LIN {X 0,Y 720.158,Z 171.461,A -85,B 0,C 180,E1 33611.893,E2 33611.893} C_VEL
LIN {X 0,Y 720.133,Z 171.461,A -85,B 0,C 180,E1 33608.963,E2 33608.963} C_VEL
LIN {X 0,Y 720.115,Z 171.46,A -85,B 0,C 180,E1 33606.555,E2 33606.555} C_VEL
LIN {X 0,Y 720.175,Z 171.461,A -85,B 0,C 180,E1 33603.874,E2 33603.874} C_VEL
LIN {X 0,Y 720.128,Z 171.46,A -85,B 0,C 180,E1 33601.001,E2 33601.001} C_VEL
LIN {X 0,Y 720.115,Z 171.461,A -85,B 0,C 180,E1 33598.618,E2 33598.618} C_VEL
LIN {X 0,Y 720.167,Z 171.46,A -85,B 0,C 180,E1 33596.02,E2 33596.02} C_VEL
LIN {X 0,Y 720.131,Z 171.461,A -85,B 0,C 180,E1 33593.134,E2 33593.134} C_VEL
LIN {X 0,Y 720.115,Z 171.461,A -85,B 0,C 180,E1 33590.734,E2 33590.734} C_VEL
LIN {X 0,Y 720.152,Z 171.461,A -85,B 0,C 180,E1 33588.201,E2 33588.201} C_VEL
LIN {X 0,Y 720.129,Z 171.461,A -85,B 0,C 180,E1 33585.203,E2 33585.203} C_VEL
LIN {X 0,Y 720.114,Z 171.461,A -85,B 0,C 180,E1 33582.834,E2 33582.834} C_VEL
LIN {X 0,Y 720.15,Z 171.461,A -85,B 0,C 180,E1 33580.316,E2 33580.316} C_VEL
LIN {X 0,Y 720.133,Z 171.462,A -85,B 0,C 180,E1 33577.338,E2 33577.338} C_VEL
LIN {X 0,Y 720.114,Z 171.461,A -85,B 0,C 180,E1 33574.938,E2 33574.938} C_VEL
LIN {X 0,Y 720.151,Z 171.462,A -85,B 0,C 180,E1 33572.387,E2 33572.387} C_VEL
LIN {X 0,Y 720.134,Z 171.462,A -85,B 0,C 180,E1 33569.443,E2 33569.443} C_VEL
LIN {X 0,Y 720.113,Z 171.462,A -85,B 0,C 180,E1 33567.056,E2 33567.056} C_VEL
LIN {X 0,Y 720.139,Z 171.461,A -85,B 0,C 180,E1 33564.583,E2 33564.583} C_VEL
LIN {X 0,Y 720.135,Z 171.461,A -85,B 0,C 180,E1 33561.538,E2 33561.538} C_VEL
LIN {X 0,Y 720.116,Z 171.461,A -85,B 0,C 180,E1 33559.036,E2 33559.036} C_VEL
LIN {X 0,Y 720.183,Z 171.461,A -85,B 0,C 180,E1 33556.35,E2 33556.35} C_VEL
LIN {X 0,Y 720.123,Z 171.461,A -85,B 0,C 180,E1 33553.465,E2 33553.465} C_VEL
LIN {X 0,Y 720.118,Z 171.461,A -85,B 0,C 180,E1 33551.043,E2 33551.043} C_VEL
LIN {X 0,Y 720.213,Z 171.46,A -85,B 0,C 180,E1 33548.245,E2 33548.245} C_VEL
LIN {X 0,Y 720.117,Z 171.461,A -85,B 0,C 180,E1 33545.433,E2 33545.433} C_VEL
LIN {X 0,Y 720.125,Z 171.46,A -85,B 0,C 180,E1 33543.001,E2 33543.001} C_VEL
LIN {X 0,Y 720.179,Z 171.46,A -85,B 0,C 180,E1 33540.108,E2 33540.108} C_VEL
LIN {X 0,Y 720.116,Z 171.461,A -85,B 0,C 180,E1 33537.44,E2 33537.44} C_VEL
LIN {X 0,Y 720.139,Z 171.461,A -85,B 0,C 180,E1 33534.918,E2 33534.918} C_VEL
LIN {X 0,Y 720.134,Z 171.461,A -85,B 0,C 180,E1 33531.845,E2 33531.845} C_VEL
LIN {X 0,Y 720.115,Z 171.46,A -85,B 0,C 180,E1 33529.422,E2 33529.422} C_VEL
LIN {X 0,Y 720.149,Z 171.461,A -85,B 0,C 180,E1 33526.914,E2 33526.914} C_VEL
LIN {X 0,Y 720.131,Z 171.46,A -85,B 0,C 180,E1 33523.902,E2 33523.902} C_VEL
LIN {X 0,Y 720.116,Z 171.46,A -85,B 0,C 180,E1 33521.436,E2 33521.436} C_VEL
LIN {X 0,Y 720.193,Z 171.46,A -85,B 0,C 180,E1 33518.725,E2 33518.725} C_VEL
LIN {X 0,Y 720.121,Z 171.453,A -85,B 0,C 180,E1 33515.87,E2 33515.87} C_VEL
LIN {X 0,Y 720.118,Z 171.457,A -85,B 0,C 180,E1 33513.449,E2 33513.449} C_VEL
LIN {X 0,Y 720.211,Z 171.457,A -85,B 0,C 180,E1 33510.611,E2 33510.611} C_VEL
LIN {X 0,Y 720.117,Z 171.447,A -85,B 0,C 180,E1 33507.827,E2 33507.827} C_VEL
LIN {X 0,Y 720.126,Z 171.457,A -85,B 0,C 180,E1 33505.407,E2 33505.407} C_VEL
LIN {X 0,Y 720.166,Z 171.457,A -85,B 0,C 180,E1 33502.446,E2 33502.446} C_VEL
LIN {X 0,Y 720.116,Z 171.46,A -85,B 0,C 180,E1 33499.888,E2 33499.888} C_VEL
LIN {X 0,Y 720.126,Z 171.458,A -85,B 0,C 180,E1 33497.491,E2 33497.491} C_VEL
LIN {X 0,Y 720.167,Z 171.459,A -85,B 0,C 180,E1 33494.555,E2 33494.555} C_VEL
LIN {X 0,Y 720.115,Z 171.457,A -85,B 0,C 180,E1 33491.94,E2 33491.94} C_VEL
LIN {X 0,Y 720.14,Z 171.46,A -85,B 0,C 180,E1 33489.43,E2 33489.43} C_VEL
LIN {X 0,Y 720.136,Z 171.459,A -85,B 0,C 180,E1 33486.377,E2 33486.377} C_VEL
LIN {X 0,Y 720.115,Z 171.46,A -85,B 0,C 180,E1 33483.901,E2 33483.901} C_VEL
LIN {X 0,Y 720.169,Z 171.457,A -85,B 0,C 180,E1 33481.273,E2 33481.273} C_VEL
LIN {X 0,Y 720.126,Z 171.458,A -85,B 0,C 180,E1 33478.334,E2 33478.334} C_VEL
LIN {X 0,Y 720.117,Z 171.458,A -85,B 0,C 180,E1 33475.939,E2 33475.939} C_VEL
LIN {X 0,Y 720.21,Z 171.459,A -85,B 0,C 180,E1 33473.143,E2 33473.143} C_VEL
LIN {X 0,Y 720.12,Z 171.459,A -85,B 0,C 180,E1 33470.3,E2 33470.3} C_VEL
LIN {X 0,Y 720.123,Z 171.458,A -85,B 0,C 180,E1 33467.897,E2 33467.897} C_VEL
LIN {X 0,Y 720.195,Z 171.46,A -85,B 0,C 180,E1 33465.035,E2 33465.035} C_VEL
LIN {X 0,Y 720.117,Z 171.457,A -85,B 0,C 180,E1 33462.297,E2 33462.297} C_VEL
LIN {X 0,Y 720.131,Z 171.46,A -85,B 0,C 180,E1 33459.858,E2 33459.858} C_VEL
LIN {X 0,Y 720.155,Z 171.46,A -85,B 0,C 180,E1 33456.863,E2 33456.863} C_VEL
LIN {X 0,Y 720.117,Z 171.458,A -85,B 0,C 180,E1 33454.292,E2 33454.292} C_VEL
LIN {X 0,Y 720.152,Z 171.451,A -85,B 0,C 180,E1 33451.741,E2 33451.741} C_VEL
LIN {X 0,Y 720.136,Z 171.46,A -85,B 0,C 180,E1 33448.78,E2 33448.78} C_VEL
LIN {X 0,Y 720.116,Z 171.458,A -85,B 0,C 180,E1 33446.357,E2 33446.357} C_VEL
LIN {X 0,Y 720.165,Z 171.456,A -85,B 0,C 180,E1 33443.739,E2 33443.739} C_VEL
LIN {X 0,Y 720.128,Z 171.456,A -85,B 0,C 180,E1 33440.775,E2 33440.775} C_VEL
LIN {X 0,Y 720.117,Z 171.46,A -85,B 0,C 180,E1 33438.416,E2 33438.416} C_VEL
LIN {X 0,Y 720.178,Z 171.459,A -85,B 0,C 180,E1 33435.751,E2 33435.751} C_VEL
LIN {X 0,Y 720.127,Z 171.458,A -85,B 0,C 180,E1 33432.851,E2 33432.851} C_VEL
LIN {X 0,Y 720.119,Z 171.461,A -85,B 0,C 180,E1 33430.456,E2 33430.456} C_VEL
LIN {X 0,Y 720.191,Z 171.446,A -85,B 0,C 180,E1 33427.748,E2 33427.748} C_VEL
LIN {X 0,Y 720.122,Z 171.461,A -85,B 0,C 180,E1 33424.854,E2 33424.854} C_VEL
LIN {X 0,Y 720.122,Z 171.447,A -85,B 0,C 180,E1 33422.404,E2 33422.404} C_VEL
LIN {X 0,Y 720.19,Z 171.751,A -85,B 0,C 180,E1 33421.207,E2 33421.207} C_VEL
LIN {X 0,Y 722.827,Z 180.968,A -85,B 0,C 180,E1 33420.32,E2 33420.32} C_VEL
LIN {X 0,Y 722.315,Z 216.19,A -85,B 0,C 180,E1 33417.535,E2 33417.535} C_VEL
LIN {X 0,Y 722.261,Z 226.415,A -85,B 0,C 180,E1 33416.755,E2 33416.755} C_VEL
LIN {X 0,Y 723.859,Z 234.554,A -85,B 0,C 180,E1 33416.596,E2 33416.596} C_VEL
LIN {X 0,Y 723.073,Z 507.416,A -85,B 0,C 180,E1 33413.694,E2 33413.694} C_VEL
LIN {X 0,Y 722.911,Z 536.198,A -85,B 0,C 180,E1 33413.337,E2 33413.337} C_VEL
LIN {X 0,Y 722.72,Z 557.475,A -85,B 0,C 180,E1 33412.924,E2 33412.924} C_VEL
LIN {X 0,Y 722.482,Z 576.531,A -85,B 0,C 180,E1 33412.43,E2 33412.43} C_VEL
LIN {X 0,Y 722.235,Z 596.799,A -85,B 0,C 180,E1 33411.776,E2 33411.776} C_VEL
LIN {X 0,Y 721.924,Z 617.74,A -85,B 0,C 180,E1 33410.934,E2 33410.934} C_VEL
LIN {X 0,Y 721.584,Z 636.362,A -85,B 0,C 180,E1 33410.032,E2 33410.032} C_VEL
LIN {X 0,Y 721.311,Z 654.533,A -85,B 0,C 180,E1 33409.009,E2 33409.009} C_VEL
LIN {X 0,Y 720.986,Z 673.25,A -85,B 0,C 180,E1 33407.762,E2 33407.762} C_VEL
LIN {X 0,Y 720.714,Z 689.21,A -85,B 0,C 180,E1 33406.521,E2 33406.521} C_VEL
LIN {X 0,Y 720.486,Z 704.756,A -85,B 0,C 180,E1 33405.122,E2 33405.122} C_VEL
LIN {X 0,Y 720.286,Z 719.459,A -85,B 0,C 180,E1 33403.566,E2 33403.566} C_VEL
LIN {X 0,Y 720.163,Z 731.326,A -85,B 0,C 180,E1 33402.1,E2 33402.1} C_VEL
LIN {X 0,Y 720.053,Z 742.382,A -85,B 0,C 180,E1 33400.48,E2 33400.48} C_VEL
LIN {X 0,Y 719.976,Z 751.89,A -85,B 0,C 180,E1 33398.786,E2 33398.786} C_VEL
LIN {X 0,Y 719.946,Z 759.234,A -85,B 0,C 180,E1 33397.179,E2 33397.179} C_VEL
LIN {X 0,Y 719.924,Z 765.17,A -85,B 0,C 180,E1 33395.498,E2 33395.498} C_VEL
LIN {X 0,Y 719.917,Z 769.789,A -85,B 0,C 180,E1 33393.663,E2 33393.663} C_VEL
LIN {X 0,Y 719.919,Z 772.482,A -85,B 0,C 180,E1 33391.91,E2 33391.91} C_VEL
LIN {X 0,Y 719.907,Z 773.462,A -85,B 0,C 180,E1 33390.159,E2 33390.159} C_VEL
LIN {X 0,Y 719.91,Z 772.697,A -85,B 0,C 180,E1 33388.329,E2 33388.329} C_VEL
LIN {X 0,Y 719.908,Z 770.262,A -85,B 0,C 180,E1 33386.577,E2 33386.577} C_VEL
LIN {X 0,Y 719.909,Z 766.362,A -85,B 0,C 180,E1 33384.901,E2 33384.901} C_VEL
LIN {X 0,Y 719.925,Z 760.484,A -85,B 0,C 180,E1 33383.141,E2 33383.141} C_VEL
LIN {X 0,Y 719.965,Z 752.702,A -85,B 0,C 180,E1 33381.375,E2 33381.375} C_VEL
LIN {X 0,Y 720.041,Z 743.892,A -85,B 0,C 180,E1 33379.763,E2 33379.763} C_VEL
LIN {X 0,Y 720.147,Z 732.537,A -85,B 0,C 180,E1 33378.062,E2 33378.062} C_VEL
LIN {X 0,Y 720.262,Z 720.869,A -85,B 0,C 180,E1 33376.597,E2 33376.597} C_VEL
LIN {X 0,Y 720.458,Z 707.3,A -85,B 0,C 180,E1 33375.125,E2 33375.125} C_VEL
LIN {X 0,Y 720.7,Z 691.197,A -85,B 0,C 180,E1 33373.644,E2 33373.644} C_VEL
LIN {X 0,Y 720.947,Z 675.482,A -85,B 0,C 180,E1 33372.404,E2 33372.404} C_VEL
LIN {X 0,Y 721.234,Z 657.839,A -85,B 0,C 180,E1 33371.199,E2 33371.199} C_VEL
LIN {X 0,Y 721.563,Z 638.343,A -85,B 0,C 180,E1 33370.072,E2 33370.072} C_VEL
LIN {X 0,Y 721.867,Z 620.585,A -85,B 0,C 180,E1 33369.196,E2 33369.196} C_VEL
LIN {X 0,Y 722.145,Z 601.277,A -85,B 0,C 180,E1 33368.392,E2 33368.392} C_VEL
LIN {X 0,Y 722.463,Z 579.414,A -85,B 0,C 180,E1 33367.654,E2 33367.654} C_VEL
LIN {X 0,Y 722.691,Z 559.421,A -85,B 0,C 180,E1 33367.121,E2 33367.121} C_VEL
LIN {X 0,Y 722.903,Z 537.995,A -85,B 0,C 180,E1 33366.692,E2 33366.692} C_VEL
LIN {X 0,Y 723.061,Z 510.848,A -85,B 0,C 180,E1 33366.342,E2 33366.342} C_VEL
LIN {X 0,Y 723.844,Z 239.48,A -85,B 0,C 180,E1 33363.457,E2 33363.457} C_VEL
LIN {X 0,Y 723.623,Z 232.466,A -85,B 0,C 180,E1 33363.372,E2 33363.372} C_VEL
LIN {X 0,Y 722.233,Z 225.971,A -85,B 0,C 180,E1 33363.219,E2 33363.219} C_VEL
LIN {X 0,Y 722.711,Z 188.921,A -85,B 0,C 180,E1 33360.315,E2 33360.315} C_VEL
LIN {X 0,Y 722.78,Z 180.457,A -85,B 0,C 180,E1 33359.636,E2 33359.636} C_VEL
LIN {X 0,Y 720.169,Z 171.589,A -85,B 0,C 180,E1 33358.76,E2 33358.76} C_VEL
LIN {X 0,Y 720.136,Z 171.461,A -85,B 0,C 180,E1 33355.788,E2 33355.788} C_VEL
LIN {X 0,Y 720.116,Z 171.457,A -85,B 0,C 180,E1 33353.346,E2 33353.346} C_VEL
LIN {X 0,Y 720.16,Z 171.454,A -85,B 0,C 180,E1 33350.782,E2 33350.782} C_VEL
LIN {X 0,Y 720.132,Z 171.458,A -85,B 0,C 180,E1 33347.855,E2 33347.855} C_VEL
LIN {X 0,Y 720.117,Z 171.46,A -85,B 0,C 180,E1 33345.423,E2 33345.423} C_VEL
LIN {X 0,Y 720.18,Z 171.458,A -85,B 0,C 180,E1 33342.747,E2 33342.747} C_VEL
LIN {X 0,Y 720.127,Z 171.456,A -85,B 0,C 180,E1 33339.849,E2 33339.849} C_VEL
LIN {X 0,Y 720.119,Z 171.46,A -85,B 0,C 180,E1 33337.428,E2 33337.428} C_VEL
LIN {X 0,Y 720.203,Z 171.454,A -85,B 0,C 180,E1 33334.696,E2 33334.696} C_VEL
LIN {X 0,Y 720.12,Z 171.46,A -85,B 0,C 180,E1 33331.827,E2 33331.827} C_VEL
LIN {X 0,Y 720.118,Z 171.455,A -85,B 0,C 180,E1 33329.486,E2 33329.486} C_VEL
LIN {X 0,Y 720.208,Z 171.452,A -85,B 0,C 180,E1 33326.732,E2 33326.732} C_VEL
LIN {X 0,Y 720.121,Z 171.46,A -85,B 0,C 180,E1 33323.919,E2 33323.919} C_VEL
LIN {X 0,Y 720.12,Z 171.457,A -85,B 0,C 180,E1 33321.539,E2 33321.539} C_VEL
LIN {X 0,Y 720.205,Z 171.457,A -85,B 0,C 180,E1 33318.706,E2 33318.706} C_VEL
LIN {X 0,Y 720.118,Z 171.459,A -85,B 0,C 180,E1 33315.958,E2 33315.958} C_VEL
LIN {X 0,Y 720.12,Z 171.458,A -85,B 0,C 180,E1 33313.634,E2 33313.634} C_VEL
LIN {X 0,Y 720.203,Z 171.46,A -85,B 0,C 180,E1 33310.803,E2 33310.803} C_VEL
LIN {X 0,Y 720.118,Z 171.456,A -85,B 0,C 180,E1 33308.062,E2 33308.062} C_VEL
LIN {X 0,Y 720.12,Z 171.46,A -85,B 0,C 180,E1 33305.738,E2 33305.738} C_VEL
LIN {X 0,Y 720.209,Z 171.457,A -85,B 0,C 180,E1 33302.945,E2 33302.945} C_VEL
LIN {X 0,Y 720.119,Z 171.46,A -85,B 0,C 180,E1 33300.159,E2 33300.159} C_VEL
LIN {X 0,Y 720.121,Z 171.457,A -85,B 0,C 180,E1 33297.772,E2 33297.772} C_VEL
LIN {X 0,Y 720.191,Z 171.459,A -85,B 0,C 180,E1 33294.902,E2 33294.902} C_VEL
LIN {X 0,Y 720.119,Z 171.458,A -85,B 0,C 180,E1 33292.26,E2 33292.26} C_VEL
LIN {X 0,Y 720.123,Z 171.46,A -85,B 0,C 180,E1 33289.837,E2 33289.837} C_VEL
LIN {X 0,Y 720.194,Z 171.46,A -85,B 0,C 180,E1 33287.002,E2 33287.002} C_VEL
LIN {X 0,Y 720.116,Z 171.459,A -85,B 0,C 180,E1 33284.29,E2 33284.29} C_VEL
LIN {X 0,Y 720.164,Z 171.459,A -85,B 0,C 180,E1 33283.499,E2 33283.499} C_VEL
LIN {X 0,Y 719.244,Z 171.582,A -85,B 0,C 180,E1 33282.887,E2 33282.887} C_VEL
LIN {X 0,Y 712.687,Z 172.397,A -85,B 0,C 180,E1 33281.126,E2 33281.126} C_VEL
LIN {X 0,Y 712.206,Z 172.449,A -85,B 0,C 180,E1 33280.724,E2 33280.724} C_VEL
LIN {X 0,Y 712.176,Z 172.446,A -85,B 0,C 180,E1 33278.244,E2 33278.244} C_VEL
LIN {X 0,Y 712.218,Z 172.449,A -85,B 0,C 180,E1 33275.646,E2 33275.646} C_VEL
LIN {X 0,Y 712.191,Z 172.435,A -85,B 0,C 180,E1 33272.671,E2 33272.671} C_VEL
LIN {X 0,Y 712.178,Z 172.446,A -85,B 0,C 180,E1 33270.29,E2 33270.29} C_VEL
LIN {X 0,Y 712.215,Z 172.449,A -85,B 0,C 180,E1 33267.758,E2 33267.758} C_VEL
LIN {X 0,Y 712.188,Z 172.441,A -85,B 0,C 180,E1 33264.758,E2 33264.758} C_VEL
LIN {X 0,Y 712.177,Z 172.449,A -85,B 0,C 180,E1 33262.349,E2 33262.349} C_VEL
LIN {X 0,Y 712.242,Z 172.449,A -85,B 0,C 180,E1 33259.658,E2 33259.658} C_VEL
LIN {X 0,Y 712.184,Z 172.45,A -85,B 0,C 180,E1 33256.753,E2 33256.753} C_VEL
LIN {X 0,Y 712.178,Z 172.45,A -85,B 0,C 180,E1 33254.354,E2 33254.354} C_VEL
LIN {X 0,Y 712.273,Z 172.449,A -85,B 0,C 180,E1 33251.563,E2 33251.563} C_VEL
LIN {X 0,Y 712.18,Z 172.45,A -85,B 0,C 180,E1 33248.762,E2 33248.762} C_VEL
LIN {X 0,Y 712.185,Z 172.449,A -85,B 0,C 180,E1 33246.304,E2 33246.304} C_VEL
LIN {X 0,Y 712.233,Z 172.45,A -85,B 0,C 180,E1 33243.352,E2 33243.352} C_VEL
LIN {X 0,Y 712.176,Z 172.45,A -85,B 0,C 180,E1 33240.729,E2 33240.729} C_VEL
LIN {X 0,Y 712.19,Z 172.45,A -85,B 0,C 180,E1 33238.323,E2 33238.323} C_VEL
LIN {X 0,Y 712.212,Z 172.45,A -85,B 0,C 180,E1 33235.294,E2 33235.294} C_VEL
LIN {X 0,Y 712.177,Z 172.45,A -85,B 0,C 180,E1 33232.796,E2 33232.796} C_VEL
LIN {X 0,Y 712.193,Z 172.45,A -85,B 0,C 180,E1 33230.373,E2 33230.373} C_VEL
LIN {X 0,Y 712.203,Z 172.45,A -85,B 0,C 180,E1 33227.313,E2 33227.313} C_VEL
LIN {X 0,Y 712.176,Z 172.451,A -85,B 0,C 180,E1 33224.803,E2 33224.803} C_VEL
LIN {X 0,Y 712.217,Z 172.45,A -85,B 0,C 180,E1 33222.237,E2 33222.237} C_VEL
LIN {X 0,Y 712.189,Z 172.45,A -85,B 0,C 180,E1 33219.251,E2 33219.251} C_VEL
LIN {X 0,Y 712.177,Z 172.451,A -85,B 0,C 180,E1 33216.853,E2 33216.853} C_VEL
LIN {X 0,Y 712.238,Z 172.45,A -85,B 0,C 180,E1 33214.186,E2 33214.186} C_VEL
LIN {X 0,Y 712.184,Z 172.451,A -85,B 0,C 180,E1 33211.287,E2 33211.287} C_VEL
LIN {X 0,Y 712.176,Z 172.451,A -85,B 0,C 180,E1 33208.954,E2 33208.954} C_VEL
LIN {X 0,Y 712.232,Z 172.451,A -85,B 0,C 180,E1 33206.298,E2 33206.298} C_VEL
LIN {X 0,Y 712.187,Z 172.451,A -85,B 0,C 180,E1 33203.39,E2 33203.39} C_VEL
LIN {X 0,Y 712.177,Z 172.45,A -85,B 0,C 180,E1 33201.036,E2 33201.036} C_VEL
LIN {X 0,Y 712.242,Z 172.451,A -85,B 0,C 180,E1 33198.339,E2 33198.339} C_VEL
LIN {X 0,Y 712.184,Z 172.451,A -85,B 0,C 180,E1 33195.447,E2 33195.447} C_VEL
LIN {X 0,Y 712.179,Z 172.45,A -85,B 0,C 180,E1 33193.023,E2 33193.023} C_VEL
LIN {X 0,Y 712.272,Z 172.449,A -85,B 0,C 180,E1 33190.228,E2 33190.228} C_VEL
LIN {X 0,Y 712.181,Z 172.45,A -85,B 0,C 180,E1 33187.466,E2 33187.466} C_VEL
LIN {X 0,Y 712.18,Z 172.45,A -85,B 0,C 180,E1 33185.091,E2 33185.091} C_VEL
LIN {X 0,Y 712.261,Z 172.45,A -85,B 0,C 180,E1 33182.225,E2 33182.225} C_VEL
LIN {X 0,Y 712.18,Z 172.45,A -85,B 0,C 180,E1 33179.548,E2 33179.548} C_VEL
LIN {X 0,Y 712.184,Z 172.45,A -85,B 0,C 180,E1 33177.094,E2 33177.094} C_VEL
LIN {X 0,Y 712.24,Z 172.449,A -85,B 0,C 180,E1 33174.174,E2 33174.174} C_VEL
LIN {X 0,Y 712.178,Z 172.45,A -85,B 0,C 180,E1 33171.546,E2 33171.546} C_VEL
LIN {X 0,Y 712.188,Z 172.449,A -85,B 0,C 180,E1 33169.144,E2 33169.144} C_VEL
LIN {X 0,Y 712.226,Z 172.45,A -85,B 0,C 180,E1 33166.187,E2 33166.187} C_VEL
LIN {X 0,Y 712.178,Z 172.45,A -85,B 0,C 180,E1 33163.58,E2 33163.58} C_VEL
LIN {X 0,Y 712.2,Z 172.449,A -85,B 0,C 180,E1 33161.075,E2 33161.075} C_VEL
LIN {X 0,Y 712.199,Z 172.449,A -85,B 0,C 180,E1 33158.047,E2 33158.047} C_VEL
LIN {X 0,Y 712.174,Z 172.441,A -85,B 0,C 180,E1 33155.539,E2 33155.539} C_VEL
LIN {X 0,Y 712.255,Z 172.446,A -85,B 0,C 180,E1 33152.777,E2 33152.777} C_VEL
LIN {X 0,Y 712.182,Z 172.446,A -85,B 0,C 180,E1 33149.895,E2 33149.895} C_VEL
LIN {X 0,Y 712.179,Z 172.434,A -85,B 0,C 180,E1 33147.511,E2 33147.511} C_VEL
LIN {X 0,Y 712.261,Z 172.449,A -85,B 0,C 180,E1 33144.641,E2 33144.641} C_VEL
LIN {X 0,Y 712.178,Z 172.446,A -85,B 0,C 180,E1 33141.889,E2 33141.889} C_VEL
LIN {X 0,Y 712.19,Z 172.449,A -85,B 0,C 180,E1 33139.435,E2 33139.435} C_VEL
LIN {X 0,Y 712.222,Z 172.447,A -85,B 0,C 180,E1 33136.475,E2 33136.475} C_VEL
LIN {X 0,Y 712.177,Z 172.448,A -85,B 0,C 180,E1 33133.974,E2 33133.974} C_VEL
LIN {X 0,Y 712.192,Z 172.445,A -85,B 0,C 180,E1 33131.5,E2 33131.5} C_VEL
LIN {X 0,Y 712.211,Z 172.446,A -85,B 0,C 180,E1 33128.477,E2 33128.477} C_VEL
LIN {X 0,Y 712.177,Z 172.448,A -85,B 0,C 180,E1 33126.044,E2 33126.044} C_VEL
LIN {X 0,Y 712.195,Z 172.449,A -85,B 0,C 180,E1 33123.556,E2 33123.556} C_VEL
LIN {X 0,Y 712.2,Z 172.449,A -85,B 0,C 180,E1 33120.483,E2 33120.483} C_VEL
LIN {X 0,Y 712.177,Z 172.447,A -85,B 0,C 180,E1 33118.069,E2 33118.069} C_VEL
LIN {X 0,Y 712.202,Z 172.447,A -85,B 0,C 180,E1 33115.571,E2 33115.571} C_VEL
LIN {X 0,Y 712.194,Z 172.444,A -85,B 0,C 180,E1 33112.498,E2 33112.498} C_VEL
LIN {X 0,Y 712.177,Z 172.448,A -85,B 0,C 180,E1 33110.056,E2 33110.056} C_VEL
LIN {X 0,Y 712.254,Z 172.447,A -85,B 0,C 180,E1 33107.3,E2 33107.3} C_VEL
LIN {X 0,Y 712.185,Z 172.449,A -85,B 0,C 180,E1 33104.445,E2 33104.445} C_VEL
LIN {X 0,Y 712.182,Z 172.445,A -85,B 0,C 180,E1 33102.008,E2 33102.008} C_VEL
LIN {X 0,Y 712.269,Z 172.447,A -85,B 0,C 180,E1 33099.196,E2 33099.196} C_VEL
LIN {X 0,Y 712.18,Z 172.449,A -85,B 0,C 180,E1 33096.413,E2 33096.413} C_VEL
LIN {X 0,Y 712.192,Z 172.447,A -85,B 0,C 180,E1 33093.932,E2 33093.932} C_VEL
LIN {X 0,Y 712.216,Z 172.443,A -85,B 0,C 180,E1 33090.938,E2 33090.938} C_VEL
LIN {X 0,Y 712.179,Z 172.449,A -85,B 0,C 180,E1 33088.42,E2 33088.42} C_VEL
LIN {X 0,Y 712.201,Z 172.447,A -85,B 0,C 180,E1 33085.916,E2 33085.916} C_VEL
LIN {X 0,Y 712.199,Z 172.449,A -85,B 0,C 180,E1 33082.865,E2 33082.865} C_VEL
LIN {X 0,Y 712.178,Z 172.445,A -85,B 0,C 180,E1 33080.401,E2 33080.401} C_VEL
LIN {X 0,Y 712.222,Z 172.449,A -85,B 0,C 180,E1 33077.83,E2 33077.83} C_VEL
LIN {X 0,Y 712.19,Z 172.449,A -85,B 0,C 180,E1 33074.846,E2 33074.846} C_VEL
LIN {X 0,Y 712.18,Z 172.447,A -85,B 0,C 180,E1 33072.396,E2 33072.396} C_VEL
LIN {X 0,Y 712.274,Z 172.443,A -85,B 0,C 180,E1 33069.584,E2 33069.584} C_VEL
LIN {X 0,Y 712.184,Z 172.445,A -85,B 0,C 180,E1 33066.828,E2 33066.828} C_VEL
LIN {X 0,Y 712.186,Z 172.451,A -85,B 0,C 180,E1 33064.355,E2 33064.355} C_VEL
LIN {X 0,Y 712.284,Z 172.657,A -85,B 0,C 180,E1 33061.516,E2 33061.516} C_VEL
LIN {X 0,Y 715.411,Z 184.026,A -85,B 0,C 180,E1 33060.418,E2 33060.418} C_VEL
LIN {X 0,Y 714.784,Z 219.598,A -85,B 0,C 180,E1 33057.578,E2 33057.578} C_VEL
LIN {X 0,Y 714.793,Z 226.685,A -85,B 0,C 180,E1 33057.05,E2 33057.05} C_VEL
LIN {X 0,Y 716.697,Z 236.047,A -85,B 0,C 180,E1 33056.867,E2 33056.867} C_VEL
LIN {X 0,Y 715.741,Z 508.433,A -85,B 0,C 180,E1 33053.941,E2 33053.941} C_VEL
LIN {X 0,Y 715.55,Z 536.813,A -85,B 0,C 180,E1 33053.582,E2 33053.582} C_VEL
LIN {X 0,Y 715.315,Z 557.949,A -85,B 0,C 180,E1 33053.163,E2 33053.163} C_VEL
LIN {X 0,Y 715.033,Z 576.766,A -85,B 0,C 180,E1 33052.669,E2 33052.669} C_VEL
LIN {X 0,Y 714.713,Z 597.931,A -85,B 0,C 180,E1 33051.974,E2 33051.974} C_VEL
LIN {X 0,Y 714.335,Z 618.643,A -85,B 0,C 180,E1 33051.124,E2 33051.124} C_VEL
LIN {X 0,Y 713.968,Z 635.93,A -85,B 0,C 180,E1 33050.278,E2 33050.278} C_VEL
LIN {X 0,Y 713.632,Z 653.828,A -85,B 0,C 180,E1 33049.264,E2 33049.264} C_VEL
LIN {X 0,Y 713.223,Z 673.243,A -85,B 0,C 180,E1 33047.962,E2 33047.962} C_VEL
LIN {X 0,Y 712.903,Z 688.705,A -85,B 0,C 180,E1 33046.749,E2 33046.749} C_VEL
LIN {X 0,Y 712.633,Z 703.912,A -85,B 0,C 180,E1 33045.376,E2 33045.376} C_VEL
LIN {X 0,Y 712.387,Z 719.074,A -85,B 0,C 180,E1 33043.765,E2 33043.765} C_VEL
LIN {X 0,Y 712.218,Z 731.015,A -85,B 0,C 180,E1 33042.278,E2 33042.278} C_VEL
LIN {X 0,Y 712.086,Z 741.867,A -85,B 0,C 180,E1 33040.68,E2 33040.68} C_VEL
LIN {X 0,Y 712,Z 751.485,A -85,B 0,C 180,E1 33038.967,E2 33038.967} C_VEL
LIN {X 0,Y 711.949,Z 758.898,A -85,B 0,C 180,E1 33037.342,E2 33037.342} C_VEL
LIN {X 0,Y 711.925,Z 764.919,A -85,B 0,C 180,E1 33035.641,E2 33035.641} C_VEL
LIN {X 0,Y 711.919,Z 769.632,A -85,B 0,C 180,E1 33033.784,E2 33033.784} C_VEL
LIN {X 0,Y 711.913,Z 772.302,A -85,B 0,C 180,E1 33032.092,E2 33032.092} C_VEL
LIN {X 0,Y 711.899,Z 773.396,A -85,B 0,C 180,E1 33030.402,E2 33030.402} C_VEL
LIN {X 0,Y 711.899,Z 772.9,A -85,B 0,C 180,E1 33028.551,E2 33028.551} C_VEL
LIN {X 0,Y 711.9,Z 770.702,A -85,B 0,C 180,E1 33026.78,E2 33026.78} C_VEL
LIN {X 0,Y 711.904,Z 767.182,A -85,B 0,C 180,E1 33025.167,E2 33025.167} C_VEL
LIN {X 0,Y 711.928,Z 761.697,A -85,B 0,C 180,E1 33023.388,E2 33023.388} C_VEL
LIN {X 0,Y 711.971,Z 754.288,A -85,B 0,C 180,E1 33021.603,E2 33021.603} C_VEL
LIN {X 0,Y 712.048,Z 746.209,A -85,B 0,C 180,E1 33020.055,E2 33020.055} C_VEL
LIN {X 0,Y 712.154,Z 736.005,A -85,B 0,C 180,E1 33018.419,E2 33018.419} C_VEL
LIN {X 0,Y 712.315,Z 723.655,A -85,B 0,C 180,E1 33016.775,E2 33016.775} C_VEL
LIN {X 0,Y 712.508,Z 711.24,A -85,B 0,C 180,E1 33015.371,E2 33015.371} C_VEL
LIN {X 0,Y 712.764,Z 696.584,A -85,B 0,C 180,E1 33013.935,E2 33013.935} C_VEL
LIN {X 0,Y 713.087,Z 679.358,A -85,B 0,C 180,E1 33012.499,E2 33012.499} C_VEL
LIN {X 0,Y 713.429,Z 663.221,A -85,B 0,C 180,E1 33011.341,E2 33011.341} C_VEL
LIN {X 0,Y 713.783,Z 645.985,A -85,B 0,C 180,E1 33010.272,E2 33010.272} C_VEL
LIN {X 0,Y 714.194,Z 625.031,A -85,B 0,C 180,E1 33009.172,E2 33009.172} C_VEL
LIN {X 0,Y 714.565,Z 605.599,A -85,B 0,C 180,E1 33008.324,E2 33008.324} C_VEL
LIN {X 0,Y 714.906,Z 586.052,A -85,B 0,C 180,E1 33007.616,E2 33007.616} C_VEL
LIN {X 0,Y 715.254,Z 562.564,A -85,B 0,C 180,E1 33006.945,E2 33006.945} C_VEL
LIN {X 0,Y 715.502,Z 541.455,A -85,B 0,C 180,E1 33006.5,E2 33006.5} C_VEL
LIN {X 0,Y 715.668,Z 520.882,A -85,B 0,C 180,E1 33006.197,E2 33006.197} C_VEL
LIN {X 0,Y 716.645,Z 251.057,A -85,B 0,C 180,E1 33003.296,E2 33003.296} C_VEL
LIN {X 0,Y 716.483,Z 233.974,A -85,B 0,C 180,E1 33003.102,E2 33003.102} C_VEL
LIN {X 0,Y 714.725,Z 225.985,A -85,B 0,C 180,E1 33002.915,E2 33002.915} C_VEL
LIN {X 0,Y 715.316,Z 189.489,A -85,B 0,C 180,E1 33000.023,E2 33000.023} C_VEL
LIN {X 0,Y 715.181,Z 182.609,A -85,B 0,C 180,E1 32999.455,E2 32999.455} C_VEL
LIN {X 0,Y 712.275,Z 172.574,A -85,B 0,C 180,E1 32998.466,E2 32998.466} C_VEL
LIN {X 0,Y 712.186,Z 172.45,A -85,B 0,C 180,E1 32995.643,E2 32995.643} C_VEL
LIN {X 0,Y 712.183,Z 172.445,A -85,B 0,C 180,E1 32993.156,E2 32993.156} C_VEL
LIN {X 0,Y 712.256,Z 172.449,A -85,B 0,C 180,E1 32990.292,E2 32990.292} C_VEL
LIN {X 0,Y 712.18,Z 172.447,A -85,B 0,C 180,E1 32987.604,E2 32987.604} C_VEL
LIN {X 0,Y 712.191,Z 172.449,A -85,B 0,C 180,E1 32985.154,E2 32985.154} C_VEL
LIN {X 0,Y 712.22,Z 172.449,A -85,B 0,C 180,E1 32982.15,E2 32982.15} C_VEL
LIN {X 0,Y 712.177,Z 172.445,A -85,B 0,C 180,E1 32979.585,E2 32979.585} C_VEL
LIN {X 0,Y 712.2,Z 172.449,A -85,B 0,C 180,E1 32977.124,E2 32977.124} C_VEL
LIN {X 0,Y 712.2,Z 172.447,A -85,B 0,C 180,E1 32974.068,E2 32974.068} C_VEL
LIN {X 0,Y 712.179,Z 172.449,A -85,B 0,C 180,E1 32971.559,E2 32971.559} C_VEL
LIN {X 0,Y 712.229,Z 172.443,A -85,B 0,C 180,E1 32968.97,E2 32968.97} C_VEL
LIN {X 0,Y 712.191,Z 172.447,A -85,B 0,C 180,E1 32966.05,E2 32966.05} C_VEL
LIN {X 0,Y 712.182,Z 172.449,A -85,B 0,C 180,E1 32963.556,E2 32963.556} C_VEL
LIN {X 0,Y 712.271,Z 172.448,A -85,B 0,C 180,E1 32960.718,E2 32960.718} C_VEL
LIN {X 0,Y 712.179,Z 172.445,A -85,B 0,C 180,E1 32957.907,E2 32957.907} C_VEL
LIN {X 0,Y 712.19,Z 172.448,A -85,B 0,C 180,E1 32955.471,E2 32955.471} C_VEL
LIN {X 0,Y 712.219,Z 172.447,A -85,B 0,C 180,E1 32952.486,E2 32952.486} C_VEL
LIN {X 0,Y 712.177,Z 172.448,A -85,B 0,C 180,E1 32949.863,E2 32949.863} C_VEL
LIN {X 0,Y 712.222,Z 172.444,A -85,B 0,C 180,E1 32947.259,E2 32947.259} C_VEL
LIN {X 0,Y 712.188,Z 172.447,A -85,B 0,C 180,E1 32944.267,E2 32944.267} C_VEL
LIN {X 0,Y 712.18,Z 172.447,A -85,B 0,C 180,E1 32941.812,E2 32941.812} C_VEL
LIN {X 0,Y 712.273,Z 172.447,A -85,B 0,C 180,E1 32939.035,E2 32939.035} C_VEL
LIN {X 0,Y 712.179,Z 172.449,A -85,B 0,C 180,E1 32936.216,E2 32936.216} C_VEL
LIN {X 0,Y 712.184,Z 172.448,A -85,B 0,C 180,E1 32933.794,E2 32933.794} C_VEL
LIN {X 0,Y 712.255,Z 172.449,A -85,B 0,C 180,E1 32930.954,E2 32930.954} C_VEL
LIN {X 0,Y 712.178,Z 172.446,A -85,B 0,C 180,E1 32928.254,E2 32928.254} C_VEL
LIN {X 0,Y 712.19,Z 172.449,A -85,B 0,C 180,E1 32925.777,E2 32925.777} C_VEL
LIN {X 0,Y 712.214,Z 172.447,A -85,B 0,C 180,E1 32922.769,E2 32922.769} C_VEL
LIN {X 0,Y 712.206,Z 172.449,A -85,B 0,C 180,E1 32920.724,E2 32920.724} C_VEL
LIN {X 0,Y 711.162,Z 172.579,A -85,B 0,C 180,E1 32920.105,E2 32920.105} C_VEL
LIN {X 0,Y 704.748,Z 173.373,A -85,B 0,C 180,E1 32918.368,E2 32918.368} C_VEL
LIN {X 0,Y 704.249,Z 173.435,A -85,B 0,C 180,E1 32917.917,E2 32917.917} C_VEL
LIN {X 0,Y 704.281,Z 173.434,A -85,B 0,C 180,E1 32914.913,E2 32914.913} C_VEL
LIN {X 0,Y 704.237,Z 173.422,A -85,B 0,C 180,E1 32912.336,E2 32912.336} C_VEL
LIN {X 0,Y 704.256,Z 173.434,A -85,B 0,C 180,E1 32909.922,E2 32909.922} C_VEL
LIN {X 0,Y 704.264,Z 173.434,A -85,B 0,C 180,E1 32906.865,E2 32906.865} C_VEL
LIN {X 0,Y 704.236,Z 173.429,A -85,B 0,C 180,E1 32904.294,E2 32904.294} C_VEL
LIN {X 0,Y 704.33,Z 173.439,A -85,B 0,C 180,E1 32901.454,E2 32901.454} C_VEL
LIN {X 0,Y 704.244,Z 173.438,A -85,B 0,C 180,E1 32898.675,E2 32898.675} C_VEL
LIN {X 0,Y 704.244,Z 173.439,A -85,B 0,C 180,E1 32896.255,E2 32896.255} C_VEL
LIN {X 0,Y 704.315,Z 173.439,A -85,B 0,C 180,E1 32893.375,E2 32893.375} C_VEL
LIN {X 0,Y 704.241,Z 173.438,A -85,B 0,C 180,E1 32890.663,E2 32890.663} C_VEL
LIN {X 0,Y 704.249,Z 173.439,A -85,B 0,C 180,E1 32888.239,E2 32888.239} C_VEL
LIN {X 0,Y 704.285,Z 173.439,A -85,B 0,C 180,E1 32885.279,E2 32885.279} C_VEL
LIN {X 0,Y 704.238,Z 173.439,A -85,B 0,C 180,E1 32882.647,E2 32882.647} C_VEL
LIN {X 0,Y 704.273,Z 173.439,A -85,B 0,C 180,E1 32880.073,E2 32880.073} C_VEL
LIN {X 0,Y 704.256,Z 173.439,A -85,B 0,C 180,E1 32877.101,E2 32877.101} C_VEL
LIN {X 0,Y 704.238,Z 173.44,A -85,B 0,C 180,E1 32874.669,E2 32874.669} C_VEL
LIN {X 0,Y 704.311,Z 173.439,A -85,B 0,C 180,E1 32871.921,E2 32871.921} C_VEL
LIN {X 0,Y 704.245,Z 173.44,A -85,B 0,C 180,E1 32869.057,E2 32869.057} C_VEL
LIN {X 0,Y 704.244,Z 173.439,A -85,B 0,C 180,E1 32866.579,E2 32866.579} C_VEL
LIN {X 0,Y 704.316,Z 173.439,A -85,B 0,C 180,E1 32863.713,E2 32863.713} C_VEL
LIN {X 0,Y 704.239,Z 173.44,A -85,B 0,C 180,E1 32860.966,E2 32860.966} C_VEL
LIN {X 0,Y 704.263,Z 173.439,A -85,B 0,C 180,E1 32858.408,E2 32858.408} C_VEL
LIN {X 0,Y 704.258,Z 173.44,A -85,B 0,C 180,E1 32855.376,E2 32855.376} C_VEL
LIN {X 0,Y 704.238,Z 173.44,A -85,B 0,C 180,E1 32852.848,E2 32852.848} C_VEL
LIN {X 0,Y 704.342,Z 173.437,A -85,B 0,C 180,E1 32850,E2 32850} C_VEL
LIN {X 0,Y 704.238,Z 173.44,A -85,B 0,C 180,E1 32847.152,E2 32847.152} C_VEL
LIN {X 0,Y 704.257,Z 173.44,A -85,B 0,C 180,E1 32844.624,E2 32844.624} C_VEL
LIN {X 0,Y 704.255,Z 173.439,A -85,B 0,C 180,E1 32841.51,E2 32841.51} C_VEL
LIN {X 0,Y 704.239,Z 173.44,A -85,B 0,C 180,E1 32839.034,E2 32839.034} C_VEL
LIN {X 0,Y 704.329,Z 173.439,A -85,B 0,C 180,E1 32836.204,E2 32836.204} C_VEL
LIN {X 0,Y 704.241,Z 173.439,A -85,B 0,C 180,E1 32833.336,E2 32833.336} C_VEL
LIN {X 0,Y 704.251,Z 173.44,A -85,B 0,C 180,E1 32830.857,E2 32830.857} C_VEL
LIN {X 0,Y 704.271,Z 173.439,A -85,B 0,C 180,E1 32827.815,E2 32827.815} C_VEL
LIN {X 0,Y 704.239,Z 173.439,A -85,B 0,C 180,E1 32825.242,E2 32825.242} C_VEL
LIN {X 0,Y 704.303,Z 173.439,A -85,B 0,C 180,E1 32822.527,E2 32822.527} C_VEL
LIN {X 0,Y 704.247,Z 173.439,A -85,B 0,C 180,E1 32819.643,E2 32819.643} C_VEL
LIN {X 0,Y 704.242,Z 173.439,A -85,B 0,C 180,E1 32817.16,E2 32817.16} C_VEL
LIN {X 0,Y 704.318,Z 173.439,A -85,B 0,C 180,E1 32814.296,E2 32814.296} C_VEL
LIN {X 0,Y 704.239,Z 173.439,A -85,B 0,C 180,E1 32811.553,E2 32811.553} C_VEL
LIN {X 0,Y 704.25,Z 173.438,A -85,B 0,C 180,E1 32809.123,E2 32809.123} C_VEL
LIN {X 0,Y 704.283,Z 173.439,A -85,B 0,C 180,E1 32806.153,E2 32806.153} C_VEL
LIN {X 0,Y 704.24,Z 173.439,A -85,B 0,C 180,E1 32803.614,E2 32803.614} C_VEL
LIN {X 0,Y 704.261,Z 173.439,A -85,B 0,C 180,E1 32801.08,E2 32801.08} C_VEL
LIN {X 0,Y 704.257,Z 173.438,A -85,B 0,C 180,E1 32798.013,E2 32798.013} C_VEL
LIN {X 0,Y 704.237,Z 173.429,A -85,B 0,C 180,E1 32795.5,E2 32795.5} C_VEL
LIN {X 0,Y 704.326,Z 173.436,A -85,B 0,C 180,E1 32792.647,E2 32792.647} C_VEL
LIN {X 0,Y 704.243,Z 173.434,A -85,B 0,C 180,E1 32789.844,E2 32789.844} C_VEL
LIN {X 0,Y 704.242,Z 173.421,A -85,B 0,C 180,E1 32787.469,E2 32787.469} C_VEL
LIN {X 0,Y 704.312,Z 173.438,A -85,B 0,C 180,E1 32784.58,E2 32784.58} C_VEL
LIN {X 0,Y 704.238,Z 173.435,A -85,B 0,C 180,E1 32781.839,E2 32781.839} C_VEL
LIN {X 0,Y 704.262,Z 173.438,A -85,B 0,C 180,E1 32779.318,E2 32779.318} C_VEL
LIN {X 0,Y 704.256,Z 173.436,A -85,B 0,C 180,E1 32776.242,E2 32776.242} C_VEL
LIN {X 0,Y 704.238,Z 173.437,A -85,B 0,C 180,E1 32773.8,E2 32773.8} C_VEL
LIN {X 0,Y 704.31,Z 173.434,A -85,B 0,C 180,E1 32771.049,E2 32771.049} C_VEL
LIN {X 0,Y 704.245,Z 173.435,A -85,B 0,C 180,E1 32768.162,E2 32768.162} C_VEL
LIN {X 0,Y 704.24,Z 173.437,A -85,B 0,C 180,E1 32765.786,E2 32765.786} C_VEL
LIN {X 0,Y 704.326,Z 173.433,A -85,B 0,C 180,E1 32762.929,E2 32762.929} C_VEL
LIN {X 0,Y 704.241,Z 173.438,A -85,B 0,C 180,E1 32760.163,E2 32760.163} C_VEL
LIN {X 0,Y 704.248,Z 173.436,A -85,B 0,C 180,E1 32757.722,E2 32757.722} C_VEL
LIN {X 0,Y 704.293,Z 173.437,A -85,B 0,C 180,E1 32754.787,E2 32754.787} C_VEL
LIN {X 0,Y 704.238,Z 173.432,A -85,B 0,C 180,E1 32752.166,E2 32752.166} C_VEL
LIN {X 0,Y 704.266,Z 173.437,A -85,B 0,C 180,E1 32749.612,E2 32749.612} C_VEL
LIN {X 0,Y 704.254,Z 173.436,A -85,B 0,C 180,E1 32746.535,E2 32746.535} C_VEL
LIN {X 0,Y 704.239,Z 173.438,A -85,B 0,C 180,E1 32744.181,E2 32744.181} C_VEL
LIN {X 0,Y 704.285,Z 173.434,A -85,B 0,C 180,E1 32741.543,E2 32741.543} C_VEL
LIN {X 0,Y 704.252,Z 173.435,A -85,B 0,C 180,E1 32738.599,E2 32738.599} C_VEL
LIN {X 0,Y 704.239,Z 173.438,A -85,B 0,C 180,E1 32736.22,E2 32736.22} C_VEL
LIN {X 0,Y 704.318,Z 173.433,A -85,B 0,C 180,E1 32733.436,E2 32733.436} C_VEL
LIN {X 0,Y 704.244,Z 173.432,A -85,B 0,C 180,E1 32730.577,E2 32730.577} C_VEL
LIN {X 0,Y 704.242,Z 173.438,A -85,B 0,C 180,E1 32728.214,E2 32728.214} C_VEL
LIN {X 0,Y 704.327,Z 173.43,A -85,B 0,C 180,E1 32725.399,E2 32725.399} C_VEL
LIN {X 0,Y 704.243,Z 173.438,A -85,B 0,C 180,E1 32722.578,E2 32722.578} C_VEL
LIN {X 0,Y 704.248,Z 173.433,A -85,B 0,C 180,E1 32720.175,E2 32720.175} C_VEL
LIN {X 0,Y 704.303,Z 173.436,A -85,B 0,C 180,E1 32717.265,E2 32717.265} C_VEL
LIN {X 0,Y 704.241,Z 173.438,A -85,B 0,C 180,E1 32714.645,E2 32714.645} C_VEL
LIN {X 0,Y 704.253,Z 173.436,A -85,B 0,C 180,E1 32712.172,E2 32712.172} C_VEL
LIN {X 0,Y 704.276,Z 173.43,A -85,B 0,C 180,E1 32709.175,E2 32709.175} C_VEL
LIN {X 0,Y 704.239,Z 173.434,A -85,B 0,C 180,E1 32706.601,E2 32706.601} C_VEL
LIN {X 0,Y 704.293,Z 173.422,A -85,B 0,C 180,E1 32703.908,E2 32703.908} C_VEL
LIN {X 0,Y 704.342,Z 173.637,A -85,B 0,C 180,E1 32701.812,E2 32701.812} C_VEL
LIN {X 0,Y 707.992,Z 186.596,A -85,B 0,C 180,E1 32700.554,E2 32700.554} C_VEL
LIN {X 0,Y 707.268,Z 222.439,A -85,B 0,C 180,E1 32697.668,E2 32697.668} C_VEL
LIN {X 0,Y 707.274,Z 226.531,A -85,B 0,C 180,E1 32697.365,E2 32697.365} C_VEL
LIN {X 0,Y 709.552,Z 237.446,A -85,B 0,C 180,E1 32697.144,E2 32697.144} C_VEL
LIN {X 0,Y 708.422,Z 509.706,A -85,B 0,C 180,E1 32694.19,E2 32694.19} C_VEL
LIN {X 0,Y 708.199,Z 537.745,A -85,B 0,C 180,E1 32693.826,E2 32693.826} C_VEL
LIN {X 0,Y 707.919,Z 558.617,A -85,B 0,C 180,E1 32693.402,E2 32693.402} C_VEL
LIN {X 0,Y 707.594,Z 577.344,A -85,B 0,C 180,E1 32692.904,E2 32692.904} C_VEL
LIN {X 0,Y 707.192,Z 599.352,A -85,B 0,C 180,E1 32692.165,E2 32692.165} C_VEL
LIN {X 0,Y 706.755,Z 619.546,A -85,B 0,C 180,E1 32691.318,E2 32691.318} C_VEL
LIN {X 0,Y 706.336,Z 636.727,A -85,B 0,C 180,E1 32690.463,E2 32690.463} C_VEL
LIN {X 0,Y 705.937,Z 654.525,A -85,B 0,C 180,E1 32689.439,E2 32689.439} C_VEL
LIN {X 0,Y 705.462,Z 673.554,A -85,B 0,C 180,E1 32688.142,E2 32688.142} C_VEL
LIN {X 0,Y 705.085,Z 689.194,A -85,B 0,C 180,E1 32686.898,E2 32686.898} C_VEL
LIN {X 0,Y 704.775,Z 703.916,A -85,B 0,C 180,E1 32685.551,E2 32685.551} C_VEL
LIN {X 0,Y 704.486,Z 718.753,A -85,B 0,C 180,E1 32683.96,E2 32683.96} C_VEL
LIN {X 0,Y 704.274,Z 730.697,A -85,B 0,C 180,E1 32682.461,E2 32682.461} C_VEL
LIN {X 0,Y 704.121,Z 741.352,A -85,B 0,C 180,E1 32680.885,E2 32680.885} C_VEL
LIN {X 0,Y 704.016,Z 751.486,A -85,B 0,C 180,E1 32679.069,E2 32679.069} C_VEL
LIN {X 0,Y 703.955,Z 758.891,A -85,B 0,C 180,E1 32677.426,E2 32677.426} C_VEL
LIN {X 0,Y 703.927,Z 764.921,A -85,B 0,C 180,E1 32675.706,E2 32675.706} C_VEL
LIN {X 0,Y 703.92,Z 769.634,A -85,B 0,C 180,E1 32673.827,E2 32673.827} C_VEL
LIN {X 0,Y 703.912,Z 772.296,A -85,B 0,C 180,E1 32672.116,E2 32672.116} C_VEL
LIN {X 0,Y 703.899,Z 773.396,A -85,B 0,C 180,E1 32670.407,E2 32670.407} C_VEL
LIN {X 0,Y 703.899,Z 772.903,A -85,B 0,C 180,E1 32668.535,E2 32668.535} C_VEL
LIN {X 0,Y 703.901,Z 770.697,A -85,B 0,C 180,E1 32666.743,E2 32666.743} C_VEL
LIN {X 0,Y 703.905,Z 767.385,A -85,B 0,C 180,E1 32665.193,E2 32665.193} C_VEL
LIN {X 0,Y 703.934,Z 762.301,A -85,B 0,C 180,E1 32663.476,E2 32663.476} C_VEL
LIN {X 0,Y 703.982,Z 754.678,A -85,B 0,C 180,E1 32661.589,E2 32661.589} C_VEL
LIN {X 0,Y 704.075,Z 746.206,A -85,B 0,C 180,E1 32659.941,E2 32659.941} C_VEL
LIN {X 0,Y 704.199,Z 736.009,A -85,B 0,C 180,E1 32658.287,E2 32658.287} C_VEL
LIN {X 0,Y 704.39,Z 723.649,A -85,B 0,C 180,E1 32656.624,E2 32656.624} C_VEL
LIN {X 0,Y 704.622,Z 711.233,A -85,B 0,C 180,E1 32655.203,E2 32655.203} C_VEL
LIN {X 0,Y 704.928,Z 696.861,A -85,B 0,C 180,E1 32653.776,E2 32653.776} C_VEL
LIN {X 0,Y 705.32,Z 679.362,A -85,B 0,C 180,E1 32652.3,E2 32652.3} C_VEL
LIN {X 0,Y 705.714,Z 662.972,A -85,B 0,C 180,E1 32651.113,E2 32651.113} C_VEL
LIN {X 0,Y 706.155,Z 645.262,A -85,B 0,C 180,E1 32650.007,E2 32650.007} C_VEL
LIN {X 0,Y 706.623,Z 625.037,A -85,B 0,C 180,E1 32648.939,E2 32648.939} C_VEL
LIN {X 0,Y 707.029,Z 606.639,A -85,B 0,C 180,E1 32648.124,E2 32648.124} C_VEL
LIN {X 0,Y 707.405,Z 588.109,A -85,B 0,C 180,E1 32647.437,E2 32647.437} C_VEL
LIN {X 0,Y 707.83,Z 565.205,A -85,B 0,C 180,E1 32646.757,E2 32646.757} C_VEL
LIN {X 0,Y 708.113,Z 544.08,A -85,B 0,C 180,E1 32646.29,E2 32646.29} C_VEL
LIN {X 0,Y 708.318,Z 524.59,A -85,B 0,C 180,E1 32645.983,E2 32645.983} C_VEL
LIN {X 0,Y 709.482,Z 254.111,A -85,B 0,C 180,E1 32643.039,E2 32643.039} C_VEL
LIN {X 0,Y 709.346,Z 235.452,A -85,B 0,C 180,E1 32642.825,E2 32642.825} C_VEL
LIN {X 0,Y 707.239,Z 226.016,A -85,B 0,C 180,E1 32642.607,E2 32642.607} C_VEL
LIN {X 0,Y 707.931,Z 190.047,A -85,B 0,C 180,E1 32639.724,E2 32639.724} C_VEL
LIN {X 0,Y 707.809,Z 185.439,A -85,B 0,C 180,E1 32639.343,E2 32639.343} C_VEL
LIN {X 0,Y 704.332,Z 173.58,A -85,B 0,C 180,E1 32638.175,E2 32638.175} C_VEL
LIN {X 0,Y 704.24,Z 173.44,A -85,B 0,C 180,E1 32635.436,E2 32635.436} C_VEL
LIN {X 0,Y 704.265,Z 173.425,A -85,B 0,C 180,E1 32632.892,E2 32632.892} C_VEL
LIN {X 0,Y 704.259,Z 173.44,A -85,B 0,C 180,E1 32629.873,E2 32629.873} C_VEL
LIN {X 0,Y 704.24,Z 173.436,A -85,B 0,C 180,E1 32627.378,E2 32627.378} C_VEL
LIN {X 0,Y 704.326,Z 173.433,A -85,B 0,C 180,E1 32624.556,E2 32624.556} C_VEL
LIN {X 0,Y 704.243,Z 173.438,A -85,B 0,C 180,E1 32621.693,E2 32621.693} C_VEL
LIN {X 0,Y 704.247,Z 173.433,A -85,B 0,C 180,E1 32619.289,E2 32619.289} C_VEL
LIN {X 0,Y 704.308,Z 173.433,A -85,B 0,C 180,E1 32616.401,E2 32616.401} C_VEL
LIN {X 0,Y 704.239,Z 173.436,A -85,B 0,C 180,E1 32613.706,E2 32613.706} C_VEL
LIN {X 0,Y 704.269,Z 173.438,A -85,B 0,C 180,E1 32611.117,E2 32611.117} C_VEL
LIN {X 0,Y 704.259,Z 173.426,A -85,B 0,C 180,E1 32608.123,E2 32608.123} C_VEL
LIN {X 0,Y 704.24,Z 173.436,A -85,B 0,C 180,E1 32605.65,E2 32605.65} C_VEL
LIN {X 0,Y 704.313,Z 173.438,A -85,B 0,C 180,E1 32602.892,E2 32602.892} C_VEL
LIN {X 0,Y 704.244,Z 173.438,A -85,B 0,C 180,E1 32599.985,E2 32599.985} C_VEL
LIN {X 0,Y 704.248,Z 173.433,A -85,B 0,C 180,E1 32597.518,E2 32597.518} C_VEL
LIN {X 0,Y 704.294,Z 173.436,A -85,B 0,C 180,E1 32594.554,E2 32594.554} C_VEL
LIN {X 0,Y 704.239,Z 173.436,A -85,B 0,C 180,E1 32591.881,E2 32591.881} C_VEL
LIN {X 0,Y 704.284,Z 173.437,A -85,B 0,C 180,E1 32589.232,E2 32589.232} C_VEL
LIN {X 0,Y 704.251,Z 173.438,A -85,B 0,C 180,E1 32586.276,E2 32586.276} C_VEL
LIN {X 0,Y 704.239,Z 173.436,A -85,B 0,C 180,E1 32583.826,E2 32583.826} C_VEL
LIN {X 0,Y 704.334,Z 173.437,A -85,B 0,C 180,E1 32580.976,E2 32580.976} C_VEL
LIN {X 0,Y 704.242,Z 173.433,A -85,B 0,C 180,E1 32578.21,E2 32578.21} C_VEL
LIN {X 0,Y 704.245,Z 173.438,A -85,B 0,C 180,E1 32575.766,E2 32575.766} C_VEL
LIN {X 0,Y 704.298,Z 173.435,A -85,B 0,C 180,E1 32572.823,E2 32572.823} C_VEL
LIN {X 0,Y 704.238,Z 173.438,A -85,B 0,C 180,E1 32570.136,E2 32570.136} C_VEL
LIN {X 0,Y 704.275,Z 173.434,A -85,B 0,C 180,E1 32567.537,E2 32567.537} C_VEL
LIN {X 0,Y 704.249,Z 173.437,A -85,B 0,C 180,E1 32564.519,E2 32564.519} C_VEL
LIN {X 0,Y 704.242,Z 173.436,A -85,B 0,C 180,E1 32562.016,E2 32562.016} C_VEL
LIN {X 0,Y 704.32,Z 173.434,A -85,B 0,C 180,E1 32559.125,E2 32559.125} C_VEL
LIN {X 0,Y 704.249,Z 173.435,A -85,B 0,C 180,E1 32557.917,E2 32557.917} C_VEL
LIN {X 0,Y 703.319,Z 173.562,A -85,B 0,C 180,E1 32557.291,E2 32557.291} C_VEL
LIN {X 0,Y 696.852,Z 174.369,A -85,B 0,C 180,E1 32555.49,E2 32555.49} C_VEL
LIN {X 0,Y 696.367,Z 174.423,A -85,B 0,C 180,E1 32555.079,E2 32555.079} C_VEL
LIN {X 0,Y 696.298,Z 174.409,A -85,B 0,C 180,E1 32552.362,E2 32552.362} C_VEL
LIN {X 0,Y 696.317,Z 174.423,A -85,B 0,C 180,E1 32549.924,E2 32549.924} C_VEL
LIN {X 0,Y 696.322,Z 174.423,A -85,B 0,C 180,E1 32546.83,E2 32546.83} C_VEL
LIN {X 0,Y 696.3,Z 174.416,A -85,B 0,C 180,E1 32544.235,E2 32544.235} C_VEL
LIN {X 0,Y 696.388,Z 174.427,A -85,B 0,C 180,E1 32541.348,E2 32541.348} C_VEL
LIN {X 0,Y 696.301,Z 174.427,A -85,B 0,C 180,E1 32538.546,E2 32538.546} C_VEL
LIN {X 0,Y 696.324,Z 174.428,A -85,B 0,C 180,E1 32535.998,E2 32535.998} C_VEL
LIN {X 0,Y 696.313,Z 174.428,A -85,B 0,C 180,E1 32532.887,E2 32532.887} C_VEL
LIN {X 0,Y 696.301,Z 174.428,A -85,B 0,C 180,E1 32530.44,E2 32530.44} C_VEL
LIN {X 0,Y 696.391,Z 174.427,A -85,B 0,C 180,E1 32527.6,E2 32527.6} C_VEL
LIN {X 0,Y 696.301,Z 174.428,A -85,B 0,C 180,E1 32524.751,E2 32524.751} C_VEL
LIN {X 0,Y 696.322,Z 174.428,A -85,B 0,C 180,E1 32522.186,E2 32522.186} C_VEL
LIN {X 0,Y 696.321,Z 174.429,A -85,B 0,C 180,E1 32519.126,E2 32519.126} C_VEL
LIN {X 0,Y 696.3,Z 174.428,A -85,B 0,C 180,E1 32516.614,E2 32516.614} C_VEL
LIN {X 0,Y 696.387,Z 174.427,A -85,B 0,C 180,E1 32513.792,E2 32513.792} C_VEL
LIN {X 0,Y 696.304,Z 174.429,A -85,B 0,C 180,E1 32510.948,E2 32510.948} C_VEL
LIN {X 0,Y 696.314,Z 174.429,A -85,B 0,C 180,E1 32508.413,E2 32508.413} C_VEL
LIN {X 0,Y 696.323,Z 174.429,A -85,B 0,C 180,E1 32505.318,E2 32505.318} C_VEL
LIN {X 0,Y 696.3,Z 174.428,A -85,B 0,C 180,E1 32502.825,E2 32502.825} C_VEL
LIN {X 0,Y 696.365,Z 174.429,A -85,B 0,C 180,E1 32500.088,E2 32500.088} C_VEL
LIN {X 0,Y 696.306,Z 174.429,A -85,B 0,C 180,E1 32497.176,E2 32497.176} C_VEL
LIN {X 0,Y 696.305,Z 174.429,A -85,B 0,C 180,E1 32494.694,E2 32494.694} C_VEL
LIN {X 0,Y 696.356,Z 174.429,A -85,B 0,C 180,E1 32491.728,E2 32491.728} C_VEL
LIN {X 0,Y 696.3,Z 174.429,A -85,B 0,C 180,E1 32489.095,E2 32489.095} C_VEL
LIN {X 0,Y 696.323,Z 174.43,A -85,B 0,C 180,E1 32486.543,E2 32486.543} C_VEL
LIN {X 0,Y 696.317,Z 174.429,A -85,B 0,C 180,E1 32483.487,E2 32483.487} C_VEL
LIN {X 0,Y 696.3,Z 174.428,A -85,B 0,C 180,E1 32480.996,E2 32480.996} C_VEL
LIN {X 0,Y 696.389,Z 174.427,A -85,B 0,C 180,E1 32478.153,E2 32478.153} C_VEL
LIN {X 0,Y 696.304,Z 174.429,A -85,B 0,C 180,E1 32475.363,E2 32475.363} C_VEL
LIN {X 0,Y 696.309,Z 174.428,A -85,B 0,C 180,E1 32472.882,E2 32472.882} C_VEL
LIN {X 0,Y 696.346,Z 174.429,A -85,B 0,C 180,E1 32469.899,E2 32469.899} C_VEL
LIN {X 0,Y 696.301,Z 174.428,A -85,B 0,C 180,E1 32467.28,E2 32467.28} C_VEL
LIN {X 0,Y 696.339,Z 174.429,A -85,B 0,C 180,E1 32464.669,E2 32464.669} C_VEL
LIN {X 0,Y 696.312,Z 174.429,A -85,B 0,C 180,E1 32461.674,E2 32461.674} C_VEL
LIN {X 0,Y 696.3,Z 174.428,A -85,B 0,C 180,E1 32459.26,E2 32459.26} C_VEL
LIN {X 0,Y 696.385,Z 174.427,A -85,B 0,C 180,E1 32456.446,E2 32456.446} C_VEL
LIN {X 0,Y 696.306,Z 174.428,A -85,B 0,C 180,E1 32453.631,E2 32453.631} C_VEL
LIN {X 0,Y 696.308,Z 174.428,A -85,B 0,C 180,E1 32451.139,E2 32451.139} C_VEL
LIN {X 0,Y 696.351,Z 174.428,A -85,B 0,C 180,E1 32448.179,E2 32448.179} C_VEL
LIN {X 0,Y 696.298,Z 174.428,A -85,B 0,C 180,E1 32445.519,E2 32445.519} C_VEL
LIN {X 0,Y 696.341,Z 174.428,A -85,B 0,C 180,E1 32442.893,E2 32442.893} C_VEL
LIN {X 0,Y 696.314,Z 174.428,A -85,B 0,C 180,E1 32439.932,E2 32439.932} C_VEL
LIN {X 0,Y 696.301,Z 174.427,A -85,B 0,C 180,E1 32437.439,E2 32437.439} C_VEL
LIN {X 0,Y 696.381,Z 174.414,A -85,B 0,C 180,E1 32434.552,E2 32434.552} C_VEL
LIN {X 0,Y 696.302,Z 174.428,A -85,B 0,C 180,E1 32431.789,E2 32431.789} C_VEL
LIN {X 0,Y 696.31,Z 174.423,A -85,B 0,C 180,E1 32429.364,E2 32429.364} C_VEL
LIN {X 0,Y 696.34,Z 174.423,A -85,B 0,C 180,E1 32426.34,E2 32426.34} C_VEL
LIN {X 0,Y 696.301,Z 174.427,A -85,B 0,C 180,E1 32423.708,E2 32423.708} C_VEL
LIN {X 0,Y 696.356,Z 174.423,A -85,B 0,C 180,E1 32421.037,E2 32421.037} C_VEL
LIN {X 0,Y 696.307,Z 174.425,A -85,B 0,C 180,E1 32418.07,E2 32418.07} C_VEL
LIN {X 0,Y 696.308,Z 174.425,A -85,B 0,C 180,E1 32415.546,E2 32415.546} C_VEL
LIN {X 0,Y 696.356,Z 174.422,A -85,B 0,C 180,E1 32412.607,E2 32412.607} C_VEL
LIN {X 0,Y 696.3,Z 174.427,A -85,B 0,C 180,E1 32409.923,E2 32409.923} C_VEL
LIN {X 0,Y 696.335,Z 174.424,A -85,B 0,C 180,E1 32407.342,E2 32407.342} C_VEL
LIN {X 0,Y 696.315,Z 174.427,A -85,B 0,C 180,E1 32404.365,E2 32404.365} C_VEL
LIN {X 0,Y 696.3,Z 174.422,A -85,B 0,C 180,E1 32401.893,E2 32401.893} C_VEL
LIN {X 0,Y 696.387,Z 174.427,A -85,B 0,C 180,E1 32399.095,E2 32399.095} C_VEL
LIN {X 0,Y 696.302,Z 174.424,A -85,B 0,C 180,E1 32396.212,E2 32396.212} C_VEL
LIN {X 0,Y 696.314,Z 174.426,A -85,B 0,C 180,E1 32393.735,E2 32393.735} C_VEL
LIN {X 0,Y 696.343,Z 174.426,A -85,B 0,C 180,E1 32390.745,E2 32390.745} C_VEL
LIN {X 0,Y 696.3,Z 174.425,A -85,B 0,C 180,E1 32388.15,E2 32388.15} C_VEL
LIN {X 0,Y 696.354,Z 174.425,A -85,B 0,C 180,E1 32385.447,E2 32385.447} C_VEL
LIN {X 0,Y 696.312,Z 174.422,A -85,B 0,C 180,E1 32382.535,E2 32382.535} C_VEL
LIN {X 0,Y 696.305,Z 174.427,A -85,B 0,C 180,E1 32380.015,E2 32380.015} C_VEL
LIN {X 0,Y 696.373,Z 174.427,A -85,B 0,C 180,E1 32377.1,E2 32377.1} C_VEL
LIN {X 0,Y 696.302,Z 174.425,A -85,B 0,C 180,E1 32374.38,E2 32374.38} C_VEL
LIN {X 0,Y 696.328,Z 174.414,A -85,B 0,C 180,E1 32371.808,E2 32371.808} C_VEL
LIN {X 0,Y 696.32,Z 174.427,A -85,B 0,C 180,E1 32368.776,E2 32368.776} C_VEL
LIN {X 0,Y 696.302,Z 174.424,A -85,B 0,C 180,E1 32366.236,E2 32366.236} C_VEL
LIN {X 0,Y 696.383,Z 174.427,A -85,B 0,C 180,E1 32363.322,E2 32363.322} C_VEL
LIN {X 0,Y 696.302,Z 174.422,A -85,B 0,C 180,E1 32360.575,E2 32360.575} C_VEL
LIN {X 0,Y 696.315,Z 174.427,A -85,B 0,C 180,E1 32358.108,E2 32358.108} C_VEL
LIN {X 0,Y 696.332,Z 174.427,A -85,B 0,C 180,E1 32355.05,E2 32355.05} C_VEL
LIN {X 0,Y 696.301,Z 174.424,A -85,B 0,C 180,E1 32352.551,E2 32352.551} C_VEL
LIN {X 0,Y 696.344,Z 174.43,A -85,B 0,C 180,E1 32349.934,E2 32349.934} C_VEL
LIN {X 0,Y 696.315,Z 174.413,A -85,B 0,C 180,E1 32346.984,E2 32346.984} C_VEL
LIN {X 0,Y 696.305,Z 174.429,A -85,B 0,C 180,E1 32344.451,E2 32344.451} C_VEL
LIN {X 0,Y 696.358,Z 174.621,A -85,B 0,C 180,E1 32342.12,E2 32342.12} C_VEL
LIN {X 0,Y 700.541,Z 189.254,A -85,B 0,C 180,E1 32340.677,E2 32340.677} C_VEL
LIN {X 0,Y 699.766,Z 224.637,A -85,B 0,C 180,E1 32337.811,E2 32337.811} C_VEL
LIN {X 0,Y 699.881,Z 226.959,A -85,B 0,C 180,E1 32337.67,E2 32337.67} C_VEL
LIN {X 0,Y 702.424,Z 238.728,A -85,B 0,C 180,E1 32337.428,E2 32337.428} C_VEL
LIN {X 0,Y 701.119,Z 510.723,A -85,B 0,C 180,E1 32334.447,E2 32334.447} C_VEL
LIN {X 0,Y 700.853,Z 538.444,A -85,B 0,C 180,E1 32334.078,E2 32334.078} C_VEL
LIN {X 0,Y 700.548,Z 558.562,A -85,B 0,C 180,E1 32333.664,E2 32333.664} C_VEL
LIN {X 0,Y 700.176,Z 577.182,A -85,B 0,C 180,E1 32333.165,E2 32333.165} C_VEL
LIN {X 0,Y 699.763,Z 597.97,A -85,B 0,C 180,E1 32332.468,E2 32332.468} C_VEL
LIN {X 0,Y 699.231,Z 618.614,A -85,B 0,C 180,E1 32331.603,E2 32331.603} C_VEL
LIN {X 0,Y 698.759,Z 635.975,A -85,B 0,C 180,E1 32330.736,E2 32330.736} C_VEL
LIN {X 0,Y 698.304,Z 652.317,A -85,B 0,C 180,E1 32329.796,E2 32329.796} C_VEL
LIN {X 0,Y 697.8,Z 670.966,A -85,B 0,C 180,E1 32328.546,E2 32328.546} C_VEL
LIN {X 0,Y 697.334,Z 687.695,A -85,B 0,C 180,E1 32327.221,E2 32327.221} C_VEL
LIN {X 0,Y 696.947,Z 703.07,A -85,B 0,C 180,E1 32325.816,E2 32325.816} C_VEL
LIN {X 0,Y 696.601,Z 718.048,A -85,B 0,C 180,E1 32324.206,E2 32324.206} C_VEL
LIN {X 0,Y 696.344,Z 730.075,A -85,B 0,C 180,E1 32322.689,E2 32322.689} C_VEL
LIN {X 0,Y 696.167,Z 740.837,A -85,B 0,C 180,E1 32321.095,E2 32321.095} C_VEL
LIN {X 0,Y 696.034,Z 751.081,A -85,B 0,C 180,E1 32319.257,E2 32319.257} C_VEL
LIN {X 0,Y 695.963,Z 758.555,A -85,B 0,C 180,E1 32317.594,E2 32317.594} C_VEL
LIN {X 0,Y 695.934,Z 764.67,A -85,B 0,C 180,E1 32315.854,E2 32315.854} C_VEL
LIN {X 0,Y 695.921,Z 769.636,A -85,B 0,C 180,E1 32313.872,E2 32313.872} C_VEL
LIN {X 0,Y 695.911,Z 772.29,A -85,B 0,C 180,E1 32312.141,E2 32312.141} C_VEL
LIN {X 0,Y 695.899,Z 773.396,A -85,B 0,C 180,E1 32310.412,E2 32310.412} C_VEL
LIN {X 0,Y 695.9,Z 772.906,A -85,B 0,C 180,E1 32308.518,E2 32308.518} C_VEL
LIN {X 0,Y 695.903,Z 770.692,A -85,B 0,C 180,E1 32306.706,E2 32306.706} C_VEL
LIN {X 0,Y 695.906,Z 767.382,A -85,B 0,C 180,E1 32305.138,E2 32305.138} C_VEL
LIN {X 0,Y 695.938,Z 762.564,A -85,B 0,C 180,E1 32303.484,E2 32303.484} C_VEL
LIN {X 0,Y 695.994,Z 755.068,A -85,B 0,C 180,E1 32301.575,E2 32301.575} C_VEL
LIN {X 0,Y 696.098,Z 746.666,A -85,B 0,C 180,E1 32299.909,E2 32299.909} C_VEL
LIN {X 0,Y 696.232,Z 737.105,A -85,B 0,C 180,E1 32298.319,E2 32298.319} C_VEL
LIN {X 0,Y 696.454,Z 725.024,A -85,B 0,C 180,E1 32296.637,E2 32296.637} C_VEL
LIN {X 0,Y 696.726,Z 712.013,A -85,B 0,C 180,E1 32295.117,E2 32295.117} C_VEL
LIN {X 0,Y 697.079,Z 697.638,A -85,B 0,C 180,E1 32293.662,E2 32293.662} C_VEL
LIN {X 0,Y 697.543,Z 679.908,A -85,B 0,C 180,E1 32292.139,E2 32292.139} C_VEL
LIN {X 0,Y 697.97,Z 664.43,A -85,B 0,C 180,E1 32290.997,E2 32290.997} C_VEL
LIN {X 0,Y 698.456,Z 647.362,A -85,B 0,C 180,E1 32289.904,E2 32289.904} C_VEL
LIN {X 0,Y 699.015,Z 626.822,A -85,B 0,C 180,E1 32288.786,E2 32288.786} C_VEL
LIN {X 0,Y 699.501,Z 607.68,A -85,B 0,C 180,E1 32287.921,E2 32287.921} C_VEL
LIN {X 0,Y 699.927,Z 589.333,A -85,B 0,C 180,E1 32287.227,E2 32287.227} C_VEL
LIN {X 0,Y 700.397,Z 568.522,A -85,B 0,C 180,E1 32286.583,E2 32286.583} C_VEL
LIN {X 0,Y 700.748,Z 545.66,A -85,B 0,C 180,E1 32286.056,E2 32286.056} C_VEL
LIN {X 0,Y 700.992,Z 525.924,A -85,B 0,C 180,E1 32285.735,E2 32285.735} C_VEL
LIN {X 0,Y 702.327,Z 258.945,A -85,B 0,C 180,E1 32282.796,E2 32282.796} C_VEL
LIN {X 0,Y 702.221,Z 236.921,A -85,B 0,C 180,E1 32282.543,E2 32282.543} C_VEL
LIN {X 0,Y 699.786,Z 226.208,A -85,B 0,C 180,E1 32282.3,E2 32282.3} C_VEL
LIN {X 0,Y 700.524,Z 190.129,A -85,B 0,C 180,E1 32279.395,E2 32279.395} C_VEL
LIN {X 0,Y 700.083,Z 187.237,A -85,B 0,C 180,E1 32279.135,E2 32279.135} C_VEL
LIN {X 0,Y 696.346,Z 174.554,A -85,B 0,C 180,E1 32277.864,E2 32277.864} C_VEL
LIN {X 0,Y 696.301,Z 174.429,A -85,B 0,C 180,E1 32275.349,E2 32275.349} C_VEL
LIN {X 0,Y 696.37,Z 174.403,A -85,B 0,C 180,E1 32272.564,E2 32272.564} C_VEL
LIN {X 0,Y 696.308,Z 174.43,A -85,B 0,C 180,E1 32269.686,E2 32269.686} C_VEL
LIN {X 0,Y 696.307,Z 174.424,A -85,B 0,C 180,E1 32267.224,E2 32267.224} C_VEL
LIN {X 0,Y 696.377,Z 174.421,A -85,B 0,C 180,E1 32264.361,E2 32264.361} C_VEL
LIN {X 0,Y 696.302,Z 174.427,A -85,B 0,C 180,E1 32261.578,E2 32261.578} C_VEL
LIN {X 0,Y 696.328,Z 174.422,A -85,B 0,C 180,E1 32259.037,E2 32259.037} C_VEL
LIN {X 0,Y 696.315,Z 174.422,A -85,B 0,C 180,E1 32255.967,E2 32255.967} C_VEL
LIN {X 0,Y 696.303,Z 174.424,A -85,B 0,C 180,E1 32253.465,E2 32253.465} C_VEL
LIN {X 0,Y 696.385,Z 174.42,A -85,B 0,C 180,E1 32250.55,E2 32250.55} C_VEL
LIN {X 0,Y 696.302,Z 174.414,A -85,B 0,C 180,E1 32247.815,E2 32247.815} C_VEL
LIN {X 0,Y 696.324,Z 174.425,A -85,B 0,C 180,E1 32245.24,E2 32245.24} C_VEL
LIN {X 0,Y 696.32,Z 174.423,A -85,B 0,C 180,E1 32242.17,E2 32242.17} C_VEL
LIN {X 0,Y 696.3,Z 174.427,A -85,B 0,C 180,E1 32239.722,E2 32239.722} C_VEL
LIN {X 0,Y 696.375,Z 174.421,A -85,B 0,C 180,E1 32236.947,E2 32236.947} C_VEL
LIN {X 0,Y 696.308,Z 174.424,A -85,B 0,C 180,E1 32234.13,E2 32234.13} C_VEL
LIN {X 0,Y 696.304,Z 174.424,A -85,B 0,C 180,E1 32231.682,E2 32231.682} C_VEL
LIN {X 0,Y 696.376,Z 174.421,A -85,B 0,C 180,E1 32228.755,E2 32228.755} C_VEL
LIN {X 0,Y 696.302,Z 174.427,A -85,B 0,C 180,E1 32226.017,E2 32226.017} C_VEL
LIN {X 0,Y 696.325,Z 174.425,A -85,B 0,C 180,E1 32223.458,E2 32223.458} C_VEL
LIN {X 0,Y 696.318,Z 174.427,A -85,B 0,C 180,E1 32220.411,E2 32220.411} C_VEL
LIN {X 0,Y 696.299,Z 174.422,A -85,B 0,C 180,E1 32217.943,E2 32217.943} C_VEL
LIN {X 0,Y 696.382,Z 174.427,A -85,B 0,C 180,E1 32215.14,E2 32215.14} C_VEL
LIN {X 0,Y 696.307,Z 174.424,A -85,B 0,C 180,E1 32212.325,E2 32212.325} C_VEL
LIN {X 0,Y 696.308,Z 174.427,A -85,B 0,C 180,E1 32209.827,E2 32209.827} C_VEL
LIN {X 0,Y 696.358,Z 174.427,A -85,B 0,C 180,E1 32206.887,E2 32206.887} C_VEL
LIN {X 0,Y 696.3,Z 174.426,A -85,B 0,C 180,E1 32204.252,E2 32204.252} C_VEL
LIN {X 0,Y 696.328,Z 174.425,A -85,B 0,C 180,E1 32201.671,E2 32201.671} C_VEL
LIN {X 0,Y 696.315,Z 174.423,A -85,B 0,C 180,E1 32198.609,E2 32198.609} C_VEL
LIN {X 0,Y 696.302,Z 174.427,A -85,B 0,C 180,E1 32196.112,E2 32196.112} C_VEL
LIN {X 0,Y 696.367,Z 174.423,A -85,B 0,C 180,E1 32195.079,E2 32195.079} C_VEL
LIN {X 0,Y 695.304,Z 174.551,A -85,B 0,C 180,E1 32194.445,E2 32194.445} C_VEL
LIN {X 0,Y 688.869,Z 175.336,A -85,B 0,C 180,E1 32192.669,E2 32192.669} C_VEL
LIN {X 0,Y 688.361,Z 175.396,A -85,B 0,C 180,E1 32192.207,E2 32192.207} C_VEL
LIN {X 0,Y 688.458,Z 175.412,A -85,B 0,C 180,E1 32189.351,E2 32189.351} C_VEL
LIN {X 0,Y 688.362,Z 175.411,A -85,B 0,C 180,E1 32186.476,E2 32186.476} C_VEL
LIN {X 0,Y 688.389,Z 175.404,A -85,B 0,C 180,E1 32183.851,E2 32183.851} C_VEL
LIN {X 0,Y 688.376,Z 175.417,A -85,B 0,C 180,E1 32180.813,E2 32180.813} C_VEL
LIN {X 0,Y 688.361,Z 175.417,A -85,B 0,C 180,E1 32178.408,E2 32178.408} C_VEL
LIN {X 0,Y 688.44,Z 175.417,A -85,B 0,C 180,E1 32175.601,E2 32175.601} C_VEL
LIN {X 0,Y 688.364,Z 175.417,A -85,B 0,C 180,E1 32172.693,E2 32172.693} C_VEL
LIN {X 0,Y 688.377,Z 175.417,A -85,B 0,C 180,E1 32170.153,E2 32170.153} C_VEL
LIN {X 0,Y 688.376,Z 175.417,A -85,B 0,C 180,E1 32166.975,E2 32166.975} C_VEL
LIN {X 0,Y 688.366,Z 175.417,A -85,B 0,C 180,E1 32164.4,E2 32164.4} C_VEL
LIN {X 0,Y 688.436,Z 175.416,A -85,B 0,C 180,E1 32161.508,E2 32161.508} C_VEL
LIN {X 0,Y 688.363,Z 175.418,A -85,B 0,C 180,E1 32158.828,E2 32158.828} C_VEL
LIN {X 0,Y 688.379,Z 175.417,A -85,B 0,C 180,E1 32156.293,E2 32156.293} C_VEL
LIN {X 0,Y 688.378,Z 175.418,A -85,B 0,C 180,E1 32153.153,E2 32153.153} C_VEL
LIN {X 0,Y 688.362,Z 175.418,A -85,B 0,C 180,E1 32150.666,E2 32150.666} C_VEL
LIN {X 0,Y 688.448,Z 175.416,A -85,B 0,C 180,E1 32147.843,E2 32147.843} C_VEL
LIN {X 0,Y 688.363,Z 175.419,A -85,B 0,C 180,E1 32144.982,E2 32144.982} C_VEL
LIN {X 0,Y 688.374,Z 175.417,A -85,B 0,C 180,E1 32142.498,E2 32142.498} C_VEL
LIN {X 0,Y 688.382,Z 175.418,A -85,B 0,C 180,E1 32139.361,E2 32139.361} C_VEL
LIN {X 0,Y 688.361,Z 175.419,A -85,B 0,C 180,E1 32136.84,E2 32136.84} C_VEL
LIN {X 0,Y 688.445,Z 175.417,A -85,B 0,C 180,E1 32133.997,E2 32133.997} C_VEL
LIN {X 0,Y 688.364,Z 175.418,A -85,B 0,C 180,E1 32131.165,E2 32131.165} C_VEL
LIN {X 0,Y 688.367,Z 175.418,A -85,B 0,C 180,E1 32128.752,E2 32128.752} C_VEL
LIN {X 0,Y 688.423,Z 175.417,A -85,B 0,C 180,E1 32125.836,E2 32125.836} C_VEL
LIN {X 0,Y 688.361,Z 175.419,A -85,B 0,C 180,E1 32123.16,E2 32123.16} C_VEL
LIN {X 0,Y 688.382,Z 175.418,A -85,B 0,C 180,E1 32120.639,E2 32120.639} C_VEL
LIN {X 0,Y 688.374,Z 175.417,A -85,B 0,C 180,E1 32117.502,E2 32117.502} C_VEL
LIN {X 0,Y 688.365,Z 175.418,A -85,B 0,C 180,E1 32115.007,E2 32115.007} C_VEL
LIN {X 0,Y 688.448,Z 175.416,A -85,B 0,C 180,E1 32112.157,E2 32112.157} C_VEL
LIN {X 0,Y 688.361,Z 175.418,A -85,B 0,C 180,E1 32109.302,E2 32109.302} C_VEL
LIN {X 0,Y 688.39,Z 175.418,A -85,B 0,C 180,E1 32106.732,E2 32106.732} C_VEL
LIN {X 0,Y 688.376,Z 175.417,A -85,B 0,C 180,E1 32103.665,E2 32103.665} C_VEL
LIN {X 0,Y 688.364,Z 175.418,A -85,B 0,C 180,E1 32101.151,E2 32101.151} C_VEL
LIN {X 0,Y 688.444,Z 175.416,A -85,B 0,C 180,E1 32098.285,E2 32098.285} C_VEL
LIN {X 0,Y 688.361,Z 175.417,A -85,B 0,C 180,E1 32095.448,E2 32095.448} C_VEL
LIN {X 0,Y 688.41,Z 175.417,A -85,B 0,C 180,E1 32092.728,E2 32092.728} C_VEL
LIN {X 0,Y 688.376,Z 175.417,A -85,B 0,C 180,E1 32089.821,E2 32089.821} C_VEL
LIN {X 0,Y 688.365,Z 175.417,A -85,B 0,C 180,E1 32087.293,E2 32087.293} C_VEL
LIN {X 0,Y 688.44,Z 175.417,A -85,B 0,C 180,E1 32084.399,E2 32084.399} C_VEL
LIN {X 0,Y 688.362,Z 175.417,A -85,B 0,C 180,E1 32081.585,E2 32081.585} C_VEL
LIN {X 0,Y 688.393,Z 175.417,A -85,B 0,C 180,E1 32079.015,E2 32079.015} C_VEL
LIN {X 0,Y 688.375,Z 175.404,A -85,B 0,C 180,E1 32076.006,E2 32076.006} C_VEL
LIN {X 0,Y 688.366,Z 175.411,A -85,B 0,C 180,E1 32073.403,E2 32073.403} C_VEL
LIN {X 0,Y 688.426,Z 175.411,A -85,B 0,C 180,E1 32070.458,E2 32070.458} C_VEL
LIN {X 0,Y 688.361,Z 175.395,A -85,B 0,C 180,E1 32067.793,E2 32067.793} C_VEL
LIN {X 0,Y 688.391,Z 175.411,A -85,B 0,C 180,E1 32065.188,E2 32065.188} C_VEL
LIN {X 0,Y 688.373,Z 175.412,A -85,B 0,C 180,E1 32062.099,E2 32062.099} C_VEL
LIN {X 0,Y 688.365,Z 175.416,A -85,B 0,C 180,E1 32059.606,E2 32059.606} C_VEL
LIN {X 0,Y 688.441,Z 175.412,A -85,B 0,C 180,E1 32056.713,E2 32056.713} C_VEL
LIN {X 0,Y 688.361,Z 175.415,A -85,B 0,C 180,E1 32053.953,E2 32053.953} C_VEL
LIN {X 0,Y 688.385,Z 175.411,A -85,B 0,C 180,E1 32051.388,E2 32051.388} C_VEL
LIN {X 0,Y 688.381,Z 175.412,A -85,B 0,C 180,E1 32048.352,E2 32048.352} C_VEL
LIN {X 0,Y 688.36,Z 175.415,A -85,B 0,C 180,E1 32045.92,E2 32045.92} C_VEL
LIN {X 0,Y 688.427,Z 175.416,A -85,B 0,C 180,E1 32043.164,E2 32043.164} C_VEL
LIN {X 0,Y 688.368,Z 175.416,A -85,B 0,C 180,E1 32040.25,E2 32040.25} C_VEL
LIN {X 0,Y 688.37,Z 175.413,A -85,B 0,C 180,E1 32037.752,E2 32037.752} C_VEL
LIN {X 0,Y 688.41,Z 175.415,A -85,B 0,C 180,E1 32034.75,E2 32034.75} C_VEL
LIN {X 0,Y 688.362,Z 175.409,A -85,B 0,C 180,E1 32032.152,E2 32032.152} C_VEL
LIN {X 0,Y 688.397,Z 175.415,A -85,B 0,C 180,E1 32029.539,E2 32029.539} C_VEL
LIN {X 0,Y 688.373,Z 175.414,A -85,B 0,C 180,E1 32026.476,E2 32026.476} C_VEL
LIN {X 0,Y 688.365,Z 175.416,A -85,B 0,C 180,E1 32024.041,E2 32024.041} C_VEL
LIN {X 0,Y 688.449,Z 175.414,A -85,B 0,C 180,E1 32021.19,E2 32021.19} C_VEL
LIN {X 0,Y 688.363,Z 175.412,A -85,B 0,C 180,E1 32018.349,E2 32018.349} C_VEL
LIN {X 0,Y 688.389,Z 175.416,A -85,B 0,C 180,E1 32015.79,E2 32015.79} C_VEL
LIN {X 0,Y 688.375,Z 175.401,A -85,B 0,C 180,E1 32012.677,E2 32012.677} C_VEL
LIN {X 0,Y 688.363,Z 175.408,A -85,B 0,C 180,E1 32010.213,E2 32010.213} C_VEL
LIN {X 0,Y 688.448,Z 175.415,A -85,B 0,C 180,E1 32007.38,E2 32007.38} C_VEL
LIN {X 0,Y 688.365,Z 175.41,A -85,B 0,C 180,E1 32004.565,E2 32004.565} C_VEL
LIN {X 0,Y 688.377,Z 175.417,A -85,B 0,C 180,E1 32002.056,E2 32002.056} C_VEL
LIN {X 0,Y 688.384,Z 175.416,A -85,B 0,C 180,E1 31998.916,E2 31998.916} C_VEL
LIN {X 0,Y 688.366,Z 175.414,A -85,B 0,C 180,E1 31996.325,E2 31996.325} C_VEL
LIN {X 0,Y 688.437,Z 175.413,A -85,B 0,C 180,E1 31993.385,E2 31993.385} C_VEL
LIN {X 0,Y 688.366,Z 175.419,A -85,B 0,C 180,E1 31990.691,E2 31990.691} C_VEL
LIN {X 0,Y 688.376,Z 175.401,A -85,B 0,C 180,E1 31988.203,E2 31988.203} C_VEL
LIN {X 0,Y 688.388,Z 175.418,A -85,B 0,C 180,E1 31985.108,E2 31985.108} C_VEL
LIN {X 0,Y 688.369,Z 175.442,A -85,B 0,C 180,E1 31982.505,E2 31982.505} C_VEL
LIN {X 0,Y 688.608,Z 176.566,A -85,B 0,C 180,E1 31982.318,E2 31982.318} C_VEL
LIN {X 0,Y 693.094,Z 191.913,A -85,B 0,C 180,E1 31980.802,E2 31980.802} C_VEL
LIN {X 0,Y 692.313,Z 226.128,A -85,B 0,C 180,E1 31978.023,E2 31978.023} C_VEL
LIN {X 0,Y 695.312,Z 240.31,A -85,B 0,C 180,E1 31977.714,E2 31977.714} C_VEL
LIN {X 0,Y 693.828,Z 511.868,A -85,B 0,C 180,E1 31974.709,E2 31974.709} C_VEL
LIN {X 0,Y 693.531,Z 538.539,A -85,B 0,C 180,E1 31974.346,E2 31974.346} C_VEL
LIN {X 0,Y 693.2,Z 558.19,A -85,B 0,C 180,E1 31973.939,E2 31973.939} C_VEL
LIN {X 0,Y 692.809,Z 575.684,A -85,B 0,C 180,E1 31973.471,E2 31973.471} C_VEL
LIN {X 0,Y 692.381,Z 594.282,A -85,B 0,C 180,E1 31972.856,E2 31972.856} C_VEL
LIN {X 0,Y 691.793,Z 615.845,A -85,B 0,C 180,E1 31971.981,E2 31971.981} C_VEL
LIN {X 0,Y 691.226,Z 634.305,A -85,B 0,C 180,E1 31971.064,E2 31971.064} C_VEL
LIN {X 0,Y 690.721,Z 650.252,A -85,B 0,C 180,E1 31970.15,E2 31970.15} C_VEL
LIN {X 0,Y 690.195,Z 667.343,A -85,B 0,C 180,E1 31969.021,E2 31969.021} C_VEL
LIN {X 0,Y 689.594,Z 686.196,A -85,B 0,C 180,E1 31967.551,E2 31967.551} C_VEL
LIN {X 0,Y 689.164,Z 700.407,A -85,B 0,C 180,E1 31966.259,E2 31966.259} C_VEL
LIN {X 0,Y 688.813,Z 713.57,A -85,B 0,C 180,E1 31964.886,E2 31964.886} C_VEL
LIN {X 0,Y 688.484,Z 727.588,A -85,B 0,C 180,E1 31963.178,E2 31963.178} C_VEL
LIN {X 0,Y 688.254,Z 738.709,A -85,B 0,C 180,E1 31961.564,E2 31961.564} C_VEL
LIN {X 0,Y 688.114,Z 747.587,A -85,B 0,C 180,E1 31960.041,E2 31960.041} C_VEL
LIN {X 0,Y 688.003,Z 756.503,A -85,B 0,C 180,E1 31958.187,E2 31958.187} C_VEL
LIN {X 0,Y 687.944,Z 763.092,A -85,B 0,C 180,E1 31956.425,E2 31956.425} C_VEL
LIN {X 0,Y 687.908,Z 767.585,A -85,B 0,C 180,E1 31954.835,E2 31954.835} C_VEL
LIN {X 0,Y 687.9,Z 770.979,A -85,B 0,C 180,E1 31953.166,E2 31953.166} C_VEL
LIN {X 0,Y 687.9,Z 773.107,A -85,B 0,C 180,E1 31951.249,E2 31951.249} C_VEL
LIN {X 0,Y 687.901,Z 773.349,A -85,B 0,C 180,E1 31949.417,E2 31949.417} C_VEL
LIN {X 0,Y 687.909,Z 772.109,A -85,B 0,C 180,E1 31947.668,E2 31947.668} C_VEL
LIN {X 0,Y 687.921,Z 769.004,A -85,B 0,C 180,E1 31945.749,E2 31945.749} C_VEL
LIN {X 0,Y 687.944,Z 764.159,A -85,B 0,C 180,E1 31943.91,E2 31943.91} C_VEL
LIN {X 0,Y 687.99,Z 757.558,A -85,B 0,C 180,E1 31942.065,E2 31942.065} C_VEL
LIN {X 0,Y 688.1,Z 748.509,A -85,B 0,C 180,E1 31940.128,E2 31940.128} C_VEL
LIN {X 0,Y 688.244,Z 739.245,A -85,B 0,C 180,E1 31938.521,E2 31938.521} C_VEL
LIN {X 0,Y 688.469,Z 728.225,A -85,B 0,C 180,E1 31936.907,E2 31936.907} C_VEL
LIN {X 0,Y 688.798,Z 714.306,A -85,B 0,C 180,E1 31935.195,E2 31935.195} C_VEL
LIN {X 0,Y 689.141,Z 701.291,A -85,B 0,C 180,E1 31933.827,E2 31933.827} C_VEL
LIN {X 0,Y 689.58,Z 686.693,A -85,B 0,C 180,E1 31932.492,E2 31932.492} C_VEL
LIN {X 0,Y 690.157,Z 668.558,A -85,B 0,C 180,E1 31931.066,E2 31931.066} C_VEL
LIN {X 0,Y 690.696,Z 650.96,A -85,B 0,C 180,E1 31929.893,E2 31929.893} C_VEL
LIN {X 0,Y 691.2,Z 635.108,A -85,B 0,C 180,E1 31928.979,E2 31928.979} C_VEL
LIN {X 0,Y 691.757,Z 616.762,A -85,B 0,C 180,E1 31928.063,E2 31928.063} C_VEL
LIN {X 0,Y 692.359,Z 595.523,A -85,B 0,C 180,E1 31927.188,E2 31927.188} C_VEL
LIN {X 0,Y 692.786,Z 576.68,A -85,B 0,C 180,E1 31926.559,E2 31926.559} C_VEL
LIN {X 0,Y 693.196,Z 558.417,A -85,B 0,C 180,E1 31926.067,E2 31926.067} C_VEL
LIN {X 0,Y 693.523,Z 538.953,A -85,B 0,C 180,E1 31925.662,E2 31925.662} C_VEL
LIN {X 0,Y 693.817,Z 513.647,A -85,B 0,C 180,E1 31925.311,E2 31925.311} C_VEL
LIN {X 0,Y 695.297,Z 243.064,A -85,B 0,C 180,E1 31922.316,E2 31922.316} C_VEL
LIN {X 0,Y 695.027,Z 238.011,A -85,B 0,C 180,E1 31922.247,E2 31922.247} C_VEL
LIN {X 0,Y 692.338,Z 226.199,A -85,B 0,C 180,E1 31921.975,E2 31921.975} C_VEL
LIN {X 0,Y 693.105,Z 191.408,A -85,B 0,C 180,E1 31919.157,E2 31919.157} C_VEL
LIN {X 0,Y 688.389,Z 175.572,A -85,B 0,C 180,E1 31917.556,E2 31917.556} C_VEL
LIN {X 0,Y 688.368,Z 175.418,A -85,B 0,C 180,E1 31915.155,E2 31915.155} C_VEL
LIN {X 0,Y 688.424,Z 175.39,A -85,B 0,C 180,E1 31912.198,E2 31912.198} C_VEL
LIN {X 0,Y 688.364,Z 175.419,A -85,B 0,C 180,E1 31909.518,E2 31909.518} C_VEL
LIN {X 0,Y 688.389,Z 175.413,A -85,B 0,C 180,E1 31906.954,E2 31906.954} C_VEL
LIN {X 0,Y 688.376,Z 175.414,A -85,B 0,C 180,E1 31903.857,E2 31903.857} C_VEL
LIN {X 0,Y 688.367,Z 175.416,A -85,B 0,C 180,E1 31901.334,E2 31901.334} C_VEL
LIN {X 0,Y 688.44,Z 175.416,A -85,B 0,C 180,E1 31898.435,E2 31898.435} C_VEL
LIN {X 0,Y 688.363,Z 175.41,A -85,B 0,C 180,E1 31895.721,E2 31895.721} C_VEL
LIN {X 0,Y 688.39,Z 175.413,A -85,B 0,C 180,E1 31893.103,E2 31893.103} C_VEL
LIN {X 0,Y 688.377,Z 175.408,A -85,B 0,C 180,E1 31890.05,E2 31890.05} C_VEL
LIN {X 0,Y 688.361,Z 175.401,A -85,B 0,C 180,E1 31887.605,E2 31887.605} C_VEL
LIN {X 0,Y 688.441,Z 175.414,A -85,B 0,C 180,E1 31884.819,E2 31884.819} C_VEL
LIN {X 0,Y 688.365,Z 175.412,A -85,B 0,C 180,E1 31881.92,E2 31881.92} C_VEL
LIN {X 0,Y 688.374,Z 175.416,A -85,B 0,C 180,E1 31879.429,E2 31879.429} C_VEL
LIN {X 0,Y 688.393,Z 175.415,A -85,B 0,C 180,E1 31876.367,E2 31876.367} C_VEL
LIN {X 0,Y 688.361,Z 175.413,A -85,B 0,C 180,E1 31873.867,E2 31873.867} C_VEL
LIN {X 0,Y 688.404,Z 175.413,A -85,B 0,C 180,E1 31871.223,E2 31871.223} C_VEL
LIN {X 0,Y 688.374,Z 175.41,A -85,B 0,C 180,E1 31868.268,E2 31868.268} C_VEL
LIN {X 0,Y 688.363,Z 175.416,A -85,B 0,C 180,E1 31865.807,E2 31865.807} C_VEL
LIN {X 0,Y 688.446,Z 175.41,A -85,B 0,C 180,E1 31862.914,E2 31862.914} C_VEL
LIN {X 0,Y 688.363,Z 175.416,A -85,B 0,C 180,E1 31860.083,E2 31860.083} C_VEL
LIN {X 0,Y 688.38,Z 175.41,A -85,B 0,C 180,E1 31857.586,E2 31857.586} C_VEL
LIN {X 0,Y 688.38,Z 175.415,A -85,B 0,C 180,E1 31854.499,E2 31854.499} C_VEL
LIN {X 0,Y 688.361,Z 175.413,A -85,B 0,C 180,E1 31852.068,E2 31852.068} C_VEL
LIN {X 0,Y 688.419,Z 175.416,A -85,B 0,C 180,E1 31849.37,E2 31849.37} C_VEL
LIN {X 0,Y 688.367,Z 175.416,A -85,B 0,C 180,E1 31846.39,E2 31846.39} C_VEL
LIN {X 0,Y 688.364,Z 175.415,A -85,B 0,C 180,E1 31843.979,E2 31843.979} C_VEL
LIN {X 0,Y 688.443,Z 175.416,A -85,B 0,C 180,E1 31841.102,E2 31841.102} C_VEL
LIN {X 0,Y 688.362,Z 175.412,A -85,B 0,C 180,E1 31838.349,E2 31838.349} C_VEL
LIN {X 0,Y 688.382,Z 175.416,A -85,B 0,C 180,E1 31835.819,E2 31835.819} C_VEL
LIN {X 0,Y 688.374,Z 175.396,A -85,B 0,C 180,E1 31832.677,E2 31832.677} C_VEL
LIN {X 0,Y 688.361,Z 175.396,A -85,B 0,C 180,E1 31832.207,E2 31832.207} C_VEL
LIN {X 0,Y 687.421,Z 175.52,A -85,B 0,C 180,E1 31831.566,E2 31831.566} C_VEL
LIN {X 0,Y 680.983,Z 176.336,A -85,B 0,C 180,E1 31829.723,E2 31829.723} C_VEL
LIN {X 0,Y 680.513,Z 176.402,A -85,B 0,C 180,E1 31829.302,E2 31829.302} C_VEL
LIN {X 0,Y 680.423,Z 176.399,A -85,B 0,C 180,E1 31826.418,E2 31826.418} C_VEL
LIN {X 0,Y 680.48,Z 176.392,A -85,B 0,C 180,E1 31823.621,E2 31823.621} C_VEL
LIN {X 0,Y 680.43,Z 176.406,A -85,B 0,C 180,E1 31820.702,E2 31820.702} C_VEL
LIN {X 0,Y 680.427,Z 176.406,A -85,B 0,C 180,E1 31818.265,E2 31818.265} C_VEL
LIN {X 0,Y 680.492,Z 176.406,A -85,B 0,C 180,E1 31815.322,E2 31815.322} C_VEL
LIN {X 0,Y 680.423,Z 176.406,A -85,B 0,C 180,E1 31812.523,E2 31812.523} C_VEL
LIN {X 0,Y 680.483,Z 176.406,A -85,B 0,C 180,E1 31809.781,E2 31809.781} C_VEL
LIN {X 0,Y 680.43,Z 176.406,A -85,B 0,C 180,E1 31806.832,E2 31806.832} C_VEL
LIN {X 0,Y 680.436,Z 176.407,A -85,B 0,C 180,E1 31804.245,E2 31804.245} C_VEL
LIN {X 0,Y 680.447,Z 176.406,A -85,B 0,C 180,E1 31801.143,E2 31801.143} C_VEL
LIN {X 0,Y 680.423,Z 176.407,A -85,B 0,C 180,E1 31798.62,E2 31798.62} C_VEL
LIN {X 0,Y 680.508,Z 176.406,A -85,B 0,C 180,E1 31795.749,E2 31795.749} C_VEL
LIN {X 0,Y 680.425,Z 176.407,A -85,B 0,C 180,E1 31792.87,E2 31792.87} C_VEL
LIN {X 0,Y 680.446,Z 176.407,A -85,B 0,C 180,E1 31790.288,E2 31790.288} C_VEL
LIN {X 0,Y 680.436,Z 176.407,A -85,B 0,C 180,E1 31787.177,E2 31787.177} C_VEL
LIN {X 0,Y 680.428,Z 176.408,A -85,B 0,C 180,E1 31784.639,E2 31784.639} C_VEL
LIN {X 0,Y 680.491,Z 176.406,A -85,B 0,C 180,E1 31781.698,E2 31781.698} C_VEL
LIN {X 0,Y 680.422,Z 176.407,A -85,B 0,C 180,E1 31778.96,E2 31778.96} C_VEL
LIN {X 0,Y 680.458,Z 176.408,A -85,B 0,C 180,E1 31776.326,E2 31776.326} C_VEL
LIN {X 0,Y 680.432,Z 176.408,A -85,B 0,C 180,E1 31773.285,E2 31773.285} C_VEL
LIN {X 0,Y 680.428,Z 176.408,A -85,B 0,C 180,E1 31770.758,E2 31770.758} C_VEL
LIN {X 0,Y 680.497,Z 176.406,A -85,B 0,C 180,E1 31767.895,E2 31767.895} C_VEL
LIN {X 0,Y 680.422,Z 176.407,A -85,B 0,C 180,E1 31765.094,E2 31765.094} C_VEL
LIN {X 0,Y 680.469,Z 176.407,A -85,B 0,C 180,E1 31762.402,E2 31762.402} C_VEL
LIN {X 0,Y 680.431,Z 176.408,A -85,B 0,C 180,E1 31759.417,E2 31759.417} C_VEL
LIN {X 0,Y 680.432,Z 176.406,A -85,B 0,C 180,E1 31756.836,E2 31756.836} C_VEL
LIN {X 0,Y 680.46,Z 176.407,A -85,B 0,C 180,E1 31753.79,E2 31753.79} C_VEL
LIN {X 0,Y 680.423,Z 176.407,A -85,B 0,C 180,E1 31751.141,E2 31751.141} C_VEL
LIN {X 0,Y 680.513,Z 176.405,A -85,B 0,C 180,E1 31748.271,E2 31748.271} C_VEL
LIN {X 0,Y 680.425,Z 176.407,A -85,B 0,C 180,E1 31745.429,E2 31745.429} C_VEL
LIN {X 0,Y 680.447,Z 176.406,A -85,B 0,C 180,E1 31742.81,E2 31742.81} C_VEL
LIN {X 0,Y 680.437,Z 176.406,A -85,B 0,C 180,E1 31739.737,E2 31739.737} C_VEL
LIN {X 0,Y 680.427,Z 176.407,A -85,B 0,C 180,E1 31737.168,E2 31737.168} C_VEL
LIN {X 0,Y 680.487,Z 176.405,A -85,B 0,C 180,E1 31734.203,E2 31734.203} C_VEL
LIN {X 0,Y 680.422,Z 176.407,A -85,B 0,C 180,E1 31731.465,E2 31731.465} C_VEL
LIN {X 0,Y 680.468,Z 176.406,A -85,B 0,C 180,E1 31728.794,E2 31728.794} C_VEL
LIN {X 0,Y 680.432,Z 176.406,A -85,B 0,C 180,E1 31725.817,E2 31725.817} C_VEL
LIN {X 0,Y 680.426,Z 176.406,A -85,B 0,C 180,E1 31723.335,E2 31723.335} C_VEL
LIN {X 0,Y 680.494,Z 176.406,A -85,B 0,C 180,E1 31720.39,E2 31720.39} C_VEL
LIN {X 0,Y 680.423,Z 176.405,A -85,B 0,C 180,E1 31717.631,E2 31717.631} C_VEL
LIN {X 0,Y 680.476,Z 176.388,A -85,B 0,C 180,E1 31714.862,E2 31714.862} C_VEL
LIN {X 0,Y 680.432,Z 176.406,A -85,B 0,C 180,E1 31711.939,E2 31711.939} C_VEL
LIN {X 0,Y 680.425,Z 176.4,A -85,B 0,C 180,E1 31709.491,E2 31709.491} C_VEL
LIN {X 0,Y 680.502,Z 176.388,A -85,B 0,C 180,E1 31706.625,E2 31706.625} C_VEL
LIN {X 0,Y 680.424,Z 176.405,A -85,B 0,C 180,E1 31703.836,E2 31703.836} C_VEL
LIN {X 0,Y 680.446,Z 176.401,A -85,B 0,C 180,E1 31701.282,E2 31701.282} C_VEL
LIN {X 0,Y 680.442,Z 176.402,A -85,B 0,C 180,E1 31698.24,E2 31698.24} C_VEL
LIN {X 0,Y 680.424,Z 176.403,A -85,B 0,C 180,E1 31695.688,E2 31695.688} C_VEL
LIN {X 0,Y 680.507,Z 176.398,A -85,B 0,C 180,E1 31692.819,E2 31692.819} C_VEL
LIN {X 0,Y 680.423,Z 176.405,A -85,B 0,C 180,E1 31689.986,E2 31689.986} C_VEL
LIN {X 0,Y 680.457,Z 176.401,A -85,B 0,C 180,E1 31687.345,E2 31687.345} C_VEL
LIN {X 0,Y 680.433,Z 176.405,A -85,B 0,C 180,E1 31684.298,E2 31684.298} C_VEL
LIN {X 0,Y 680.427,Z 176.398,A -85,B 0,C 180,E1 31681.768,E2 31681.768} C_VEL
LIN {X 0,Y 680.488,Z 176.402,A -85,B 0,C 180,E1 31678.821,E2 31678.821} C_VEL
LIN {X 0,Y 680.422,Z 176.402,A -85,B 0,C 180,E1 31676.04,E2 31676.04} C_VEL
LIN {X 0,Y 680.493,Z 176.404,A -85,B 0,C 180,E1 31673.249,E2 31673.249} C_VEL
LIN {X 0,Y 680.429,Z 176.404,A -85,B 0,C 180,E1 31670.356,E2 31670.356} C_VEL
LIN {X 0,Y 680.436,Z 176.402,A -85,B 0,C 180,E1 31667.783,E2 31667.783} C_VEL
LIN {X 0,Y 680.447,Z 176.405,A -85,B 0,C 180,E1 31664.662,E2 31664.662} C_VEL
LIN {X 0,Y 680.424,Z 176.4,A -85,B 0,C 180,E1 31662.114,E2 31662.114} C_VEL
LIN {X 0,Y 680.512,Z 176.403,A -85,B 0,C 180,E1 31659.261,E2 31659.261} C_VEL
LIN {X 0,Y 680.427,Z 176.405,A -85,B 0,C 180,E1 31656.44,E2 31656.44} C_VEL
LIN {X 0,Y 680.445,Z 176.402,A -85,B 0,C 180,E1 31653.842,E2 31653.842} C_VEL
LIN {X 0,Y 680.436,Z 176.396,A -85,B 0,C 180,E1 31650.703,E2 31650.703} C_VEL
LIN {X 0,Y 680.426,Z 176.405,A -85,B 0,C 180,E1 31648.259,E2 31648.259} C_VEL
LIN {X 0,Y 680.504,Z 176.393,A -85,B 0,C 180,E1 31645.345,E2 31645.345} C_VEL
LIN {X 0,Y 680.426,Z 176.406,A -85,B 0,C 180,E1 31642.507,E2 31642.507} C_VEL
LIN {X 0,Y 680.45,Z 176.399,A -85,B 0,C 180,E1 31639.937,E2 31639.937} C_VEL
LIN {X 0,Y 680.441,Z 176.402,A -85,B 0,C 180,E1 31636.897,E2 31636.897} C_VEL
LIN {X 0,Y 680.429,Z 176.406,A -85,B 0,C 180,E1 31634.303,E2 31634.303} C_VEL
LIN {X 0,Y 680.487,Z 176.405,A -85,B 0,C 180,E1 31631.336,E2 31631.336} C_VEL
LIN {X 0,Y 680.422,Z 176.394,A -85,B 0,C 180,E1 31628.642,E2 31628.642} C_VEL
LIN {X 0,Y 680.47,Z 176.399,A -85,B 0,C 180,E1 31625.938,E2 31625.938} C_VEL
LIN {X 0,Y 680.429,Z 176.371,A -85,B 0,C 180,E1 31622.932,E2 31622.932} C_VEL
LIN {X 0,Y 680.478,Z 176.743,A -85,B 0,C 180,E1 31622.729,E2 31622.729} C_VEL
LIN {X 0,Y 685.65,Z 194.514,A -85,B 0,C 180,E1 31620.934,E2 31620.934} C_VEL
LIN {X 0,Y 684.88,Z 226.298,A -85,B 0,C 180,E1 31618.338,E2 31618.338} C_VEL
LIN {X 0,Y 688.215,Z 241.644,A -85,B 0,C 180,E1 31618.009,E2 31618.009} C_VEL
LIN {X 0,Y 686.55,Z 513.268,A -85,B 0,C 180,E1 31614.972,E2 31614.972} C_VEL
LIN {X 0,Y 686.223,Z 538.722,A -85,B 0,C 180,E1 31614.618,E2 31614.618} C_VEL
LIN {X 0,Y 685.869,Z 557.817,A -85,B 0,C 180,E1 31614.22,E2 31614.22} C_VEL
LIN {X 0,Y 685.457,Z 574.929,A -85,B 0,C 180,E1 31613.761,E2 31613.761} C_VEL
LIN {X 0,Y 685.001,Z 591.783,A -85,B 0,C 180,E1 31613.207,E2 31613.207} C_VEL
LIN {X 0,Y 684.438,Z 611.154,A -85,B 0,C 180,E1 31612.442,E2 31612.442} C_VEL
LIN {X 0,Y 683.722,Z 632.31,A -85,B 0,C 180,E1 31611.418,E2 31611.418} C_VEL
LIN {X 0,Y 683.145,Z 648.824,A -85,B 0,C 180,E1 31610.473,E2 31610.473} C_VEL
LIN {X 0,Y 682.559,Z 664.82,A -85,B 0,C 180,E1 31609.42,E2 31609.42} C_VEL
LIN {X 0,Y 681.994,Z 681.506,A -85,B 0,C 180,E1 31608.155,E2 31608.155} C_VEL
LIN {X 0,Y 681.439,Z 697.743,A -85,B 0,C 180,E1 31606.712,E2 31606.712} C_VEL
LIN {X 0,Y 681.003,Z 711.214,A -85,B 0,C 180,E1 31605.322,E2 31605.322} C_VEL
LIN {X 0,Y 680.678,Z 722.936,A -85,B 0,C 180,E1 31603.938,E2 31603.938} C_VEL
LIN {X 0,Y 680.381,Z 735.446,A -85,B 0,C 180,E1 31602.216,E2 31602.216} C_VEL
LIN {X 0,Y 680.168,Z 745.731,A -85,B 0,C 180,E1 31600.502,E2 31600.502} C_VEL
LIN {X 0,Y 680.051,Z 753.476,A -85,B 0,C 180,E1 31598.965,E2 31598.965} C_VEL
LIN {X 0,Y 679.972,Z 760.806,A -85,B 0,C 180,E1 31597.179,E2 31597.179} C_VEL
LIN {X 0,Y 679.927,Z 766.555,A -85,B 0,C 180,E1 31595.315,E2 31595.315} C_VEL
LIN {X 0,Y 679.917,Z 770.244,A -85,B 0,C 180,E1 31593.625,E2 31593.625} C_VEL
LIN {X 0,Y 679.914,Z 772.712,A -85,B 0,C 180,E1 31591.769,E2 31591.769} C_VEL
LIN {X 0,Y 679.902,Z 773.44,A -85,B 0,C 180,E1 31589.747,E2 31589.747} C_VEL
LIN {X 0,Y 679.915,Z 772.452,A -85,B 0,C 180,E1 31587.978,E2 31587.978} C_VEL
LIN {X 0,Y 679.921,Z 769.952,A -85,B 0,C 180,E1 31586.206,E2 31586.206} C_VEL
LIN {X 0,Y 679.936,Z 765.433,A -85,B 0,C 180,E1 31584.262,E2 31584.262} C_VEL
LIN {X 0,Y 679.975,Z 759.531,A -85,B 0,C 180,E1 31582.481,E2 31582.481} C_VEL
LIN {X 0,Y 680.062,Z 752.289,A -85,B 0,C 180,E1 31580.779,E2 31580.779} C_VEL
LIN {X 0,Y 680.217,Z 742.913,A -85,B 0,C 180,E1 31578.985,E2 31578.985} C_VEL
LIN {X 0,Y 680.444,Z 731.901,A -85,B 0,C 180,E1 31577.268,E2 31577.268} C_VEL
LIN {X 0,Y 680.735,Z 720.813,A -85,B 0,C 180,E1 31575.798,E2 31575.798} C_VEL
LIN {X 0,Y 681.103,Z 708.069,A -85,B 0,C 180,E1 31574.331,E2 31574.331} C_VEL
LIN {X 0,Y 681.627,Z 691.86,A -85,B 0,C 180,E1 31572.74,E2 31572.74} C_VEL
LIN {X 0,Y 682.122,Z 677.325,A -85,B 0,C 180,E1 31571.516,E2 31571.516} C_VEL
LIN {X 0,Y 682.654,Z 662.309,A -85,B 0,C 180,E1 31570.405,E2 31570.405} C_VEL
LIN {X 0,Y 683.309,Z 644.547,A -85,B 0,C 180,E1 31569.263,E2 31569.263} C_VEL
LIN {X 0,Y 683.984,Z 625.009,A -85,B 0,C 180,E1 31568.207,E2 31568.207} C_VEL
LIN {X 0,Y 684.532,Z 607.203,A -85,B 0,C 180,E1 31567.393,E2 31567.393} C_VEL
LIN {X 0,Y 685.039,Z 590.541,A -85,B 0,C 180,E1 31566.748,E2 31566.748} C_VEL
LIN {X 0,Y 685.502,Z 573.444,A -85,B 0,C 180,E1 31566.195,E2 31566.195} C_VEL
LIN {X 0,Y 685.977,Z 553.018,A -85,B 0,C 180,E1 31565.664,E2 31565.664} C_VEL
LIN {X 0,Y 686.371,Z 529.703,A -85,B 0,C 180,E1 31565.238,E2 31565.238} C_VEL
LIN {X 0,Y 686.707,Z 484.935,A -85,B 0,C 180,E1 31564.713,E2 31564.713} C_VEL
LIN {X 0,Y 688.147,Z 240.424,A -85,B 0,C 180,E1 31561.974,E2 31561.974} C_VEL
LIN {X 0,Y 684.852,Z 225.835,A -85,B 0,C 180,E1 31561.636,E2 31561.636} C_VEL
LIN {X 0,Y 685.636,Z 193.995,A -85,B 0,C 180,E1 31559.021,E2 31559.021} C_VEL
LIN {X 0,Y 680.449,Z 176.566,A -85,B 0,C 180,E1 31557.237,E2 31557.237} C_VEL
LIN {X 0,Y 680.483,Z 176.407,A -85,B 0,C 180,E1 31554.63,E2 31554.63} C_VEL
LIN {X 0,Y 680.43,Z 176.39,A -85,B 0,C 180,E1 31551.681,E2 31551.681} C_VEL
LIN {X 0,Y 680.433,Z 176.408,A -85,B 0,C 180,E1 31549.169,E2 31549.169} C_VEL
LIN {X 0,Y 680.474,Z 176.406,A -85,B 0,C 180,E1 31546.177,E2 31546.177} C_VEL
LIN {X 0,Y 680.424,Z 176.403,A -85,B 0,C 180,E1 31543.451,E2 31543.451} C_VEL
LIN {X 0,Y 680.517,Z 176.395,A -85,B 0,C 180,E1 31540.577,E2 31540.577} C_VEL
LIN {X 0,Y 680.426,Z 176.406,A -85,B 0,C 180,E1 31537.685,E2 31537.685} C_VEL
LIN {X 0,Y 680.452,Z 176.398,A -85,B 0,C 180,E1 31535.069,E2 31535.069} C_VEL
LIN {X 0,Y 680.44,Z 176.405,A -85,B 0,C 180,E1 31532.03,E2 31532.03} C_VEL
LIN {X 0,Y 680.425,Z 176.396,A -85,B 0,C 180,E1 31529.561,E2 31529.561} C_VEL
LIN {X 0,Y 680.511,Z 176.39,A -85,B 0,C 180,E1 31526.719,E2 31526.719} C_VEL
LIN {X 0,Y 680.425,Z 176.405,A -85,B 0,C 180,E1 31523.836,E2 31523.836} C_VEL
LIN {X 0,Y 680.446,Z 176.4,A -85,B 0,C 180,E1 31521.282,E2 31521.282} C_VEL
LIN {X 0,Y 680.437,Z 176.399,A -85,B 0,C 180,E1 31518.152,E2 31518.152} C_VEL
LIN {X 0,Y 680.428,Z 176.404,A -85,B 0,C 180,E1 31515.6,E2 31515.6} C_VEL
LIN {X 0,Y 680.496,Z 176.4,A -85,B 0,C 180,E1 31512.705,E2 31512.705} C_VEL
LIN {X 0,Y 680.423,Z 176.404,A -85,B 0,C 180,E1 31509.9,E2 31509.9} C_VEL
LIN {X 0,Y 680.477,Z 176.398,A -85,B 0,C 180,E1 31507.175,E2 31507.175} C_VEL
LIN {X 0,Y 680.43,Z 176.403,A -85,B 0,C 180,E1 31504.214,E2 31504.214} C_VEL
LIN {X 0,Y 680.431,Z 176.402,A -85,B 0,C 180,E1 31501.684,E2 31501.684} C_VEL
LIN {X 0,Y 680.476,Z 176.399,A -85,B 0,C 180,E1 31498.737,E2 31498.737} C_VEL
LIN {X 0,Y 680.421,Z 176.405,A -85,B 0,C 180,E1 31496.04,E2 31496.04} C_VEL
LIN {X 0,Y 680.49,Z 176.403,A -85,B 0,C 180,E1 31493.249,E2 31493.249} C_VEL
LIN {X 0,Y 680.43,Z 176.405,A -85,B 0,C 180,E1 31490.356,E2 31490.356} C_VEL
LIN {X 0,Y 680.435,Z 176.4,A -85,B 0,C 180,E1 31487.783,E2 31487.783} C_VEL
LIN {X 0,Y 680.446,Z 176.404,A -85,B 0,C 180,E1 31484.663,E2 31484.663} C_VEL
LIN {X 0,Y 680.424,Z 176.403,A -85,B 0,C 180,E1 31482.114,E2 31482.114} C_VEL
LIN {X 0,Y 680.51,Z 176.401,A -85,B 0,C 180,E1 31479.261,E2 31479.261} C_VEL
LIN {X 0,Y 680.427,Z 176.405,A -85,B 0,C 180,E1 31476.44,E2 31476.44} C_VEL
LIN {X 0,Y 680.443,Z 176.4,A -85,B 0,C 180,E1 31473.842,E2 31473.842} C_VEL
LIN {X 0,Y 680.437,Z 176.4,A -85,B 0,C 180,E1 31470.703,E2 31470.703} C_VEL
LIN {X 0,Y 680.513,Z 176.402,A -85,B 0,C 180,E1 31469.302,E2 31469.302} C_VEL
LIN {X 0,Y 679.47,Z 176.541,A -85,B 0,C 180,E1 31468.654,E2 31468.654} C_VEL
LIN {X 0,Y 673.019,Z 177.325,A -85,B 0,C 180,E1 31466.836,E2 31466.836} C_VEL
LIN {X 0,Y 672.483,Z 177.388,A -85,B 0,C 180,E1 31466.364,E2 31466.364} C_VEL
LIN {X 0,Y 672.559,Z 177.38,A -85,B 0,C 180,E1 31463.51,E2 31463.51} C_VEL
LIN {X 0,Y 672.487,Z 177.395,A -85,B 0,C 180,E1 31460.588,E2 31460.588} C_VEL
LIN {X 0,Y 672.496,Z 177.395,A -85,B 0,C 180,E1 31458.119,E2 31458.119} C_VEL
LIN {X 0,Y 672.514,Z 177.396,A -85,B 0,C 180,E1 31455.041,E2 31455.041} C_VEL
LIN {X 0,Y 672.486,Z 177.395,A -85,B 0,C 180,E1 31452.449,E2 31452.449} C_VEL
LIN {X 0,Y 672.571,Z 177.394,A -85,B 0,C 180,E1 31449.62,E2 31449.62} C_VEL
LIN {X 0,Y 672.486,Z 177.395,A -85,B 0,C 180,E1 31446.701,E2 31446.701} C_VEL
LIN {X 0,Y 672.525,Z 177.396,A -85,B 0,C 180,E1 31443.983,E2 31443.983} C_VEL
LIN {X 0,Y 672.493,Z 177.395,A -85,B 0,C 180,E1 31440.956,E2 31440.956} C_VEL
LIN {X 0,Y 672.487,Z 177.396,A -85,B 0,C 180,E1 31438.504,E2 31438.504} C_VEL
LIN {X 0,Y 672.564,Z 177.394,A -85,B 0,C 180,E1 31435.631,E2 31435.631} C_VEL
LIN {X 0,Y 672.485,Z 177.396,A -85,B 0,C 180,E1 31432.801,E2 31432.801} C_VEL
LIN {X 0,Y 672.52,Z 177.396,A -85,B 0,C 180,E1 31430.175,E2 31430.175} C_VEL
LIN {X 0,Y 672.493,Z 177.396,A -85,B 0,C 180,E1 31427.119,E2 31427.119} C_VEL
LIN {X 0,Y 672.492,Z 177.397,A -85,B 0,C 180,E1 31424.548,E2 31424.548} C_VEL
LIN {X 0,Y 672.522,Z 177.397,A -85,B 0,C 180,E1 31421.49,E2 31421.49} C_VEL
LIN {X 0,Y 672.484,Z 177.396,A -85,B 0,C 180,E1 31418.808,E2 31418.808} C_VEL
LIN {X 0,Y 672.571,Z 177.393,A -85,B 0,C 180,E1 31415.965,E2 31415.965} C_VEL
LIN {X 0,Y 672.484,Z 177.397,A -85,B 0,C 180,E1 31413.068,E2 31413.068} C_VEL
LIN {X 0,Y 672.515,Z 177.397,A -85,B 0,C 180,E1 31410.426,E2 31410.426} C_VEL
LIN {X 0,Y 672.493,Z 177.397,A -85,B 0,C 180,E1 31407.359,E2 31407.359} C_VEL
LIN {X 0,Y 672.49,Z 177.396,A -85,B 0,C 180,E1 31404.797,E2 31404.797} C_VEL
LIN {X 0,Y 672.533,Z 177.395,A -85,B 0,C 180,E1 31401.795,E2 31401.795} C_VEL
LIN {X 0,Y 672.484,Z 177.397,A -85,B 0,C 180,E1 31399.117,E2 31399.117} C_VEL
LIN {X 0,Y 672.566,Z 177.395,A -85,B 0,C 180,E1 31396.241,E2 31396.241} C_VEL
LIN {X 0,Y 672.487,Z 177.396,A -85,B 0,C 180,E1 31393.326,E2 31393.326} C_VEL
LIN {X 0,Y 672.517,Z 177.397,A -85,B 0,C 180,E1 31390.64,E2 31390.64} C_VEL
LIN {X 0,Y 672.5,Z 177.396,A -85,B 0,C 180,E1 31387.631,E2 31387.631} C_VEL
LIN {X 0,Y 672.491,Z 177.396,A -85,B 0,C 180,E1 31385.026,E2 31385.026} C_VEL
LIN {X 0,Y 672.534,Z 177.396,A -85,B 0,C 180,E1 31382.023,E2 31382.023} C_VEL
LIN {X 0,Y 672.484,Z 177.395,A -85,B 0,C 180,E1 31379.341,E2 31379.341} C_VEL
LIN {X 0,Y 672.558,Z 177.395,A -85,B 0,C 180,E1 31376.516,E2 31376.516} C_VEL
LIN {X 0,Y 672.487,Z 177.395,A -85,B 0,C 180,E1 31373.551,E2 31373.551} C_VEL
LIN {X 0,Y 672.512,Z 177.396,A -85,B 0,C 180,E1 31370.906,E2 31370.906} C_VEL
LIN {X 0,Y 672.502,Z 177.395,A -85,B 0,C 180,E1 31367.896,E2 31367.896} C_VEL
LIN {X 0,Y 672.488,Z 177.396,A -85,B 0,C 180,E1 31365.293,E2 31365.293} C_VEL
LIN {X 0,Y 672.548,Z 177.395,A -85,B 0,C 180,E1 31362.337,E2 31362.337} C_VEL
LIN {X 0,Y 672.485,Z 177.395,A -85,B 0,C 180,E1 31359.633,E2 31359.633} C_VEL
LIN {X 0,Y 672.516,Z 177.394,A -85,B 0,C 180,E1 31357.024,E2 31357.024} C_VEL
LIN {X 0,Y 672.493,Z 177.388,A -85,B 0,C 180,E1 31353.948,E2 31353.948} C_VEL
LIN {X 0,Y 672.493,Z 177.395,A -85,B 0,C 180,E1 31351.359,E2 31351.359} C_VEL
LIN {X 0,Y 672.522,Z 177.368,A -85,B 0,C 180,E1 31348.313,E2 31348.313} C_VEL
LIN {X 0,Y 672.485,Z 177.388,A -85,B 0,C 180,E1 31345.638,E2 31345.638} C_VEL
LIN {X 0,Y 672.577,Z 177.39,A -85,B 0,C 180,E1 31342.739,E2 31342.739} C_VEL
LIN {X 0,Y 672.486,Z 177.394,A -85,B 0,C 180,E1 31339.816,E2 31339.816} C_VEL
LIN {X 0,Y 672.537,Z 177.391,A -85,B 0,C 180,E1 31337.09,E2 31337.09} C_VEL
LIN {X 0,Y 672.49,Z 177.393,A -85,B 0,C 180,E1 31334.114,E2 31334.114} C_VEL
LIN {X 0,Y 672.499,Z 177.388,A -85,B 0,C 180,E1 31331.492,E2 31331.492} C_VEL
LIN {X 0,Y 672.498,Z 177.389,A -85,B 0,C 180,E1 31328.292,E2 31328.292} C_VEL
LIN {X 0,Y 672.485,Z 177.392,A -85,B 0,C 180,E1 31325.803,E2 31325.803} C_VEL
LIN {X 0,Y 672.563,Z 177.386,A -85,B 0,C 180,E1 31322.897,E2 31322.897} C_VEL
LIN {X 0,Y 672.485,Z 177.394,A -85,B 0,C 180,E1 31320.085,E2 31320.085} C_VEL
LIN {X 0,Y 672.524,Z 177.391,A -85,B 0,C 180,E1 31317.403,E2 31317.403} C_VEL
LIN {X 0,Y 672.493,Z 177.393,A -85,B 0,C 180,E1 31314.368,E2 31314.368} C_VEL
LIN {X 0,Y 672.488,Z 177.386,A -85,B 0,C 180,E1 31311.88,E2 31311.88} C_VEL
LIN {X 0,Y 672.55,Z 177.391,A -85,B 0,C 180,E1 31308.943,E2 31308.943} C_VEL
LIN {X 0,Y 672.484,Z 177.391,A -85,B 0,C 180,E1 31306.15,E2 31306.15} C_VEL
LIN {X 0,Y 672.533,Z 177.394,A -85,B 0,C 180,E1 31303.501,E2 31303.501} C_VEL
LIN {X 0,Y 672.491,Z 177.394,A -85,B 0,C 180,E1 31300.481,E2 31300.481} C_VEL
LIN {X 0,Y 672.497,Z 177.389,A -85,B 0,C 180,E1 31297.903,E2 31297.903} C_VEL
LIN {X 0,Y 672.506,Z 177.391,A -85,B 0,C 180,E1 31294.741,E2 31294.741} C_VEL
LIN {X 0,Y 672.485,Z 177.376,A -85,B 0,C 180,E1 31292.168,E2 31292.168} C_VEL
LIN {X 0,Y 672.564,Z 177.39,A -85,B 0,C 180,E1 31289.241,E2 31289.241} C_VEL
LIN {X 0,Y 672.485,Z 177.39,A -85,B 0,C 180,E1 31286.419,E2 31286.419} C_VEL
LIN {X 0,Y 672.562,Z 177.387,A -85,B 0,C 180,E1 31283.532,E2 31283.532} C_VEL
LIN {X 0,Y 672.488,Z 177.387,A -85,B 0,C 180,E1 31280.629,E2 31280.629} C_VEL
LIN {X 0,Y 672.499,Z 177.394,A -85,B 0,C 180,E1 31278.119,E2 31278.119} C_VEL
LIN {X 0,Y 672.505,Z 177.394,A -85,B 0,C 180,E1 31274.95,E2 31274.95} C_VEL
LIN {X 0,Y 672.489,Z 177.391,A -85,B 0,C 180,E1 31272.334,E2 31272.334} C_VEL
LIN {X 0,Y 672.547,Z 177.382,A -85,B 0,C 180,E1 31269.367,E2 31269.367} C_VEL
LIN {X 0,Y 672.485,Z 177.379,A -85,B 0,C 180,E1 31266.591,E2 31266.591} C_VEL
LIN {X 0,Y 672.553,Z 177.358,A -85,B 0,C 180,E1 31263.776,E2 31263.776} C_VEL
LIN {X 0,Y 672.547,Z 177.688,A -85,B 0,C 180,E1 31263.062,E2 31263.062} C_VEL
LIN {X 0,Y 678.207,Z 196.655,A -85,B 0,C 180,E1 31261.109,E2 31261.109} C_VEL
LIN {X 0,Y 677.441,Z 226.136,A -85,B 0,C 180,E1 31258.677,E2 31258.677} C_VEL
LIN {X 0,Y 681.13,Z 243.158,A -85,B 0,C 180,E1 31258.306,E2 31258.306} C_VEL
LIN {X 0,Y 679.291,Z 514.158,A -85,B 0,C 180,E1 31255.248,E2 31255.248} C_VEL
LIN {X 0,Y 678.928,Z 538.969,A -85,B 0,C 180,E1 31254.894,E2 31254.894} C_VEL
LIN {X 0,Y 678.554,Z 557.445,A -85,B 0,C 180,E1 31254.506,E2 31254.506} C_VEL
LIN {X 0,Y 678.098,Z 574.915,A -85,B 0,C 180,E1 31254.035,E2 31254.035} C_VEL
LIN {X 0,Y 677.592,Z 591.766,A -85,B 0,C 180,E1 31253.476,E2 31253.476} C_VEL
LIN {X 0,Y 676.997,Z 609.743,A -85,B 0,C 180,E1 31252.762,E2 31252.762} C_VEL
LIN {X 0,Y 676.225,Z 631.081,A -85,B 0,C 180,E1 31251.737,E2 31251.737} C_VEL
LIN {X 0,Y 675.562,Z 648.104,A -85,B 0,C 180,E1 31250.759,E2 31250.759} C_VEL
LIN {X 0,Y 674.936,Z 663.552,A -85,B 0,C 180,E1 31249.738,E2 31249.738} C_VEL
LIN {X 0,Y 674.369,Z 677.914,A -85,B 0,C 180,E1 31248.657,E2 31248.657} C_VEL
LIN {X 0,Y 673.76,Z 694.101,A -85,B 0,C 180,E1 31247.264,E2 31247.264} C_VEL
LIN {X 0,Y 673.221,Z 708.984,A -85,B 0,C 180,E1 31245.754,E2 31245.754} C_VEL
LIN {X 0,Y 672.84,Z 720.841,A -85,B 0,C 180,E1 31244.367,E2 31244.367} C_VEL
LIN {X 0,Y 672.515,Z 731.894,A -85,B 0,C 180,E1 31242.885,E2 31242.885} C_VEL
LIN {X 0,Y 672.259,Z 742.916,A -85,B 0,C 180,E1 31241.147,E2 31241.147} C_VEL
LIN {X 0,Y 672.085,Z 751.889,A -85,B 0,C 180,E1 31239.418,E2 31239.418} C_VEL
LIN {X 0,Y 671.99,Z 758.865,A -85,B 0,C 180,E1 31237.781,E2 31237.781} C_VEL
LIN {X 0,Y 671.949,Z 764.677,A -85,B 0,C 180,E1 31236.064,E2 31236.064} C_VEL
LIN {X 0,Y 671.923,Z 769.64,A -85,B 0,C 180,E1 31234.01,E2 31234.01} C_VEL
LIN {X 0,Y 671.909,Z 772.272,A -85,B 0,C 180,E1 31232.217,E2 31232.217} C_VEL
LIN {X 0,Y 671.9,Z 773.369,A -85,B 0,C 180,E1 31230.512,E2 31230.512} C_VEL
LIN {X 0,Y 671.898,Z 773.048,A -85,B 0,C 180,E1 31228.636,E2 31228.636} C_VEL
LIN {X 0,Y 671.902,Z 770.968,A -85,B 0,C 180,E1 31226.759,E2 31226.759} C_VEL
LIN {X 0,Y 671.91,Z 767.58,A -85,B 0,C 180,E1 31225.049,E2 31225.049} C_VEL
LIN {X 0,Y 671.948,Z 763.081,A -85,B 0,C 180,E1 31223.422,E2 31223.422} C_VEL
LIN {X 0,Y 672.022,Z 756.51,A -85,B 0,C 180,E1 31221.617,E2 31221.617} C_VEL
LIN {X 0,Y 672.171,Z 747.584,A -85,B 0,C 180,E1 31219.719,E2 31219.719} C_VEL
LIN {X 0,Y 672.349,Z 738.695,A -85,B 0,C 180,E1 31218.159,E2 31218.159} C_VEL
LIN {X 0,Y 672.643,Z 727.595,A -85,B 0,C 180,E1 31216.506,E2 31216.506} C_VEL
LIN {X 0,Y 673.071,Z 713.567,A -85,B 0,C 180,E1 31214.757,E2 31214.757} C_VEL
LIN {X 0,Y 673.488,Z 701.273,A -85,B 0,C 180,E1 31213.44,E2 31213.44} C_VEL
LIN {X 0,Y 673.992,Z 687.67,A -85,B 0,C 180,E1 31212.163,E2 31212.163} C_VEL
LIN {X 0,Y 674.647,Z 671.531,A -85,B 0,C 180,E1 31210.838,E2 31210.838} C_VEL
LIN {X 0,Y 675.363,Z 653.062,A -85,B 0,C 180,E1 31209.552,E2 31209.552} C_VEL
LIN {X 0,Y 675.966,Z 637.748,A -85,B 0,C 180,E1 31208.632,E2 31208.632} C_VEL
LIN {X 0,Y 676.559,Z 621.96,A -85,B 0,C 180,E1 31207.804,E2 31207.804} C_VEL
LIN {X 0,Y 677.13,Z 605.504,A -85,B 0,C 180,E1 31207.059,E2 31207.059} C_VEL
LIN {X 0,Y 677.738,Z 587.617,A -85,B 0,C 180,E1 31206.375,E2 31206.375} C_VEL
LIN {X 0,Y 678.384,Z 564.984,A -85,B 0,C 180,E1 31205.678,E2 31205.678} C_VEL
LIN {X 0,Y 678.823,Z 544.801,A -85,B 0,C 180,E1 31205.217,E2 31205.217} C_VEL
LIN {X 0,Y 679.13,Z 526.894,A -85,B 0,C 180,E1 31204.916,E2 31204.916} C_VEL
LIN {X 0,Y 680.454,Z 336.393,A -85,B 0,C 180,E1 31202.751,E2 31202.751} C_VEL
LIN {X 0,Y 680.959,Z 241.429,A -85,B 0,C 180,E1 31201.666,E2 31201.666} C_VEL
LIN {X 0,Y 677.407,Z 225.699,A -85,B 0,C 180,E1 31201.301,E2 31201.301} C_VEL
LIN {X 0,Y 678.207,Z 196.655,A -85,B 0,C 180,E1 31198.89,E2 31198.89} C_VEL
LIN {X 0,Y 672.527,Z 177.542,A -85,B 0,C 180,E1 31196.906,E2 31196.906} C_VEL
LIN {X 0,Y 672.506,Z 177.388,A -85,B 0,C 180,E1 31193.83,E2 31193.83} C_VEL
LIN {X 0,Y 672.487,Z 177.382,A -85,B 0,C 180,E1 31191.253,E2 31191.253} C_VEL
LIN {X 0,Y 672.565,Z 177.386,A -85,B 0,C 180,E1 31188.359,E2 31188.359} C_VEL
LIN {X 0,Y 672.486,Z 177.395,A -85,B 0,C 180,E1 31185.536,E2 31185.536} C_VEL
LIN {X 0,Y 672.537,Z 177.391,A -85,B 0,C 180,E1 31182.8,E2 31182.8} C_VEL
LIN {X 0,Y 672.495,Z 177.387,A -85,B 0,C 180,E1 31179.854,E2 31179.854} C_VEL
LIN {X 0,Y 672.492,Z 177.395,A -85,B 0,C 180,E1 31177.312,E2 31177.312} C_VEL
LIN {X 0,Y 672.532,Z 177.389,A -85,B 0,C 180,E1 31174.297,E2 31174.297} C_VEL
LIN {X 0,Y 672.487,Z 177.394,A -85,B 0,C 180,E1 31171.559,E2 31171.559} C_VEL
LIN {X 0,Y 672.575,Z 177.37,A -85,B 0,C 180,E1 31168.698,E2 31168.698} C_VEL
LIN {X 0,Y 672.487,Z 177.391,A -85,B 0,C 180,E1 31165.827,E2 31165.827} C_VEL
LIN {X 0,Y 672.525,Z 177.394,A -85,B 0,C 180,E1 31163.111,E2 31163.111} C_VEL
LIN {X 0,Y 672.496,Z 177.394,A -85,B 0,C 180,E1 31160.088,E2 31160.088} C_VEL
LIN {X 0,Y 672.491,Z 177.387,A -85,B 0,C 180,E1 31157.568,E2 31157.568} C_VEL
LIN {X 0,Y 672.537,Z 177.39,A -85,B 0,C 180,E1 31154.552,E2 31154.552} C_VEL
LIN {X 0,Y 672.484,Z 177.391,A -85,B 0,C 180,E1 31151.841,E2 31151.841} C_VEL
LIN {X 0,Y 672.565,Z 177.39,A -85,B 0,C 180,E1 31148.981,E2 31148.981} C_VEL
LIN {X 0,Y 672.49,Z 177.394,A -85,B 0,C 180,E1 31146.146,E2 31146.146} C_VEL
LIN {X 0,Y 672.498,Z 177.391,A -85,B 0,C 180,E1 31143.58,E2 31143.58} C_VEL
LIN {X 0,Y 672.503,Z 177.394,A -85,B 0,C 180,E1 31140.426,E2 31140.426} C_VEL
LIN {X 0,Y 672.485,Z 177.387,A -85,B 0,C 180,E1 31137.87,E2 31137.87} C_VEL
LIN {X 0,Y 672.563,Z 177.393,A -85,B 0,C 180,E1 31134.968,E2 31134.968} C_VEL
LIN {X 0,Y 672.486,Z 177.39,A -85,B 0,C 180,E1 31132.224,E2 31132.224} C_VEL
LIN {X 0,Y 672.517,Z 177.394,A -85,B 0,C 180,E1 31129.549,E2 31129.549} C_VEL
LIN {X 0,Y 672.496,Z 177.393,A -85,B 0,C 180,E1 31126.472,E2 31126.472} C_VEL
LIN {X 0,Y 672.488,Z 177.392,A -85,B 0,C 180,E1 31123.945,E2 31123.945} C_VEL
LIN {X 0,Y 672.547,Z 177.394,A -85,B 0,C 180,E1 31120.984,E2 31120.984} C_VEL
LIN {X 0,Y 672.484,Z 177.389,A -85,B 0,C 180,E1 31118.27,E2 31118.27} C_VEL
LIN {X 0,Y 672.531,Z 177.394,A -85,B 0,C 180,E1 31115.586,E2 31115.586} C_VEL
LIN {X 0,Y 672.488,Z 177.37,A -85,B 0,C 180,E1 31112.553,E2 31112.553} C_VEL
LIN {X 0,Y 672.493,Z 177.389,A -85,B 0,C 180,E1 31110.028,E2 31110.028} C_VEL
LIN {X 0,Y 672.521,Z 177.388,A -85,B 0,C 180,E1 31106.975,E2 31106.975} C_VEL
LIN {X 0,Y 672.483,Z 177.388,A -85,B 0,C 180,E1 31106.364,E2 31106.364} C_VEL
LIN {X 0,Y 671.502,Z 177.512,A -85,B 0,C 180,E1 31105.708,E2 31105.708} C_VEL
LIN {X 0,Y 665.157,Z 178.295,A -85,B 0,C 180,E1 31103.868,E2 31103.868} C_VEL
LIN {X 0,Y 664.625,Z 178.37,A -85,B 0,C 180,E1 31103.39,E2 31103.39} C_VEL
LIN {X 0,Y 664.547,Z 178.384,A -85,B 0,C 180,E1 31100.513,E2 31100.513} C_VEL
LIN {X 0,Y 664.581,Z 178.384,A -85,B 0,C 180,E1 31097.871,E2 31097.871} C_VEL
LIN {X 0,Y 664.559,Z 178.385,A -85,B 0,C 180,E1 31094.874,E2 31094.874} C_VEL
LIN {X 0,Y 664.554,Z 178.384,A -85,B 0,C 180,E1 31092.246,E2 31092.246} C_VEL
LIN {X 0,Y 664.585,Z 178.385,A -85,B 0,C 180,E1 31089.184,E2 31089.184} C_VEL
LIN {X 0,Y 664.549,Z 178.384,A -85,B 0,C 180,E1 31086.459,E2 31086.459} C_VEL
LIN {X 0,Y 664.622,Z 178.383,A -85,B 0,C 180,E1 31083.508,E2 31083.508} C_VEL
LIN {X 0,Y 664.546,Z 178.384,A -85,B 0,C 180,E1 31080.664,E2 31080.664} C_VEL
LIN {X 0,Y 664.607,Z 178.384,A -85,B 0,C 180,E1 31077.894,E2 31077.894} C_VEL
LIN {X 0,Y 664.55,Z 178.386,A -85,B 0,C 180,E1 31074.912,E2 31074.912} C_VEL
LIN {X 0,Y 664.567,Z 178.385,A -85,B 0,C 180,E1 31072.278,E2 31072.278} C_VEL
LIN {X 0,Y 664.558,Z 178.386,A -85,B 0,C 180,E1 31069.145,E2 31069.145} C_VEL
LIN {X 0,Y 664.554,Z 178.385,A -85,B 0,C 180,E1 31066.519,E2 31066.519} C_VEL
LIN {X 0,Y 664.586,Z 178.384,A -85,B 0,C 180,E1 31063.484,E2 31063.484} C_VEL
LIN {X 0,Y 664.547,Z 178.387,A -85,B 0,C 180,E1 31060.751,E2 31060.751} C_VEL
LIN {X 0,Y 664.619,Z 178.383,A -85,B 0,C 180,E1 31057.781,E2 31057.781} C_VEL
LIN {X 0,Y 664.546,Z 178.386,A -85,B 0,C 180,E1 31055.006,E2 31055.006} C_VEL
LIN {X 0,Y 664.611,Z 178.384,A -85,B 0,C 180,E1 31052.155,E2 31052.155} C_VEL
LIN {X 0,Y 664.549,Z 178.386,A -85,B 0,C 180,E1 31049.224,E2 31049.224} C_VEL
LIN {X 0,Y 664.56,Z 178.387,A -85,B 0,C 180,E1 31046.636,E2 31046.636} C_VEL
LIN {X 0,Y 664.559,Z 178.387,A -85,B 0,C 180,E1 31043.435,E2 31043.435} C_VEL
LIN {X 0,Y 664.549,Z 178.385,A -85,B 0,C 180,E1 31040.911,E2 31040.911} C_VEL
LIN {X 0,Y 664.607,Z 178.385,A -85,B 0,C 180,E1 31037.931,E2 31037.931} C_VEL
LIN {X 0,Y 664.545,Z 178.386,A -85,B 0,C 180,E1 31035.182,E2 31035.182} C_VEL
LIN {X 0,Y 664.62,Z 178.384,A -85,B 0,C 180,E1 31032.311,E2 31032.311} C_VEL
LIN {X 0,Y 664.548,Z 178.385,A -85,B 0,C 180,E1 31029.37,E2 31029.37} C_VEL
LIN {X 0,Y 664.567,Z 178.385,A -85,B 0,C 180,E1 31026.787,E2 31026.787} C_VEL
LIN {X 0,Y 664.559,Z 178.384,A -85,B 0,C 180,E1 31023.654,E2 31023.654} C_VEL
LIN {X 0,Y 664.554,Z 178.386,A -85,B 0,C 180,E1 31021.026,E2 31021.026} C_VEL
LIN {X 0,Y 664.59,Z 178.385,A -85,B 0,C 180,E1 31018.027,E2 31018.027} C_VEL
LIN {X 0,Y 664.545,Z 178.385,A -85,B 0,C 180,E1 31015.343,E2 31015.343} C_VEL
LIN {X 0,Y 664.631,Z 178.382,A -85,B 0,C 180,E1 31012.451,E2 31012.451} C_VEL
LIN {X 0,Y 664.548,Z 178.384,A -85,B 0,C 180,E1 31009.579,E2 31009.579} C_VEL
LIN {X 0,Y 664.576,Z 178.384,A -85,B 0,C 180,E1 31006.924,E2 31006.924} C_VEL
LIN {X 0,Y 664.56,Z 178.384,A -85,B 0,C 180,E1 31003.896,E2 31003.896} C_VEL
LIN {X 0,Y 664.551,Z 178.384,A -85,B 0,C 180,E1 31001.34,E2 31001.34} C_VEL
LIN {X 0,Y 664.612,Z 178.383,A -85,B 0,C 180,E1 30998.397,E2 30998.397} C_VEL
LIN {X 0,Y 664.541,Z 178.367,A -85,B 0,C 180,E1 30995.612,E2 30995.612} C_VEL
LIN {X 0,Y 664.62,Z 178.377,A -85,B 0,C 180,E1 30992.767,E2 30992.767} C_VEL
LIN {X 0,Y 664.55,Z 178.377,A -85,B 0,C 180,E1 30989.87,E2 30989.87} C_VEL
LIN {X 0,Y 664.565,Z 178.356,A -85,B 0,C 180,E1 30987.242,E2 30987.242} C_VEL
LIN {X 0,Y 664.564,Z 178.383,A -85,B 0,C 180,E1 30984.158,E2 30984.158} C_VEL
LIN {X 0,Y 664.547,Z 178.378,A -85,B 0,C 180,E1 30981.608,E2 30981.608} C_VEL
LIN {X 0,Y 664.623,Z 178.38,A -85,B 0,C 180,E1 30978.69,E2 30978.69} C_VEL
LIN {X 0,Y 664.545,Z 178.381,A -85,B 0,C 180,E1 30975.803,E2 30975.803} C_VEL
LIN {X 0,Y 664.612,Z 178.381,A -85,B 0,C 180,E1 30973.042,E2 30973.042} C_VEL
LIN {X 0,Y 664.549,Z 178.383,A -85,B 0,C 180,E1 30970.052,E2 30970.052} C_VEL
LIN {X 0,Y 664.58,Z 178.378,A -85,B 0,C 180,E1 30967.347,E2 30967.347} C_VEL
LIN {X 0,Y 664.557,Z 178.383,A -85,B 0,C 180,E1 30964.314,E2 30964.314} C_VEL
LIN {X 0,Y 664.552,Z 178.375,A -85,B 0,C 180,E1 30961.724,E2 30961.724} C_VEL
LIN {X 0,Y 664.592,Z 178.379,A -85,B 0,C 180,E1 30958.707,E2 30958.707} C_VEL
LIN {X 0,Y 664.547,Z 178.379,A -85,B 0,C 180,E1 30955.945,E2 30955.945} C_VEL
LIN {X 0,Y 664.628,Z 178.374,A -85,B 0,C 180,E1 30953.001,E2 30953.001} C_VEL
LIN {X 0,Y 664.546,Z 178.382,A -85,B 0,C 180,E1 30950.123,E2 30950.123} C_VEL
LIN {X 0,Y 664.626,Z 178.375,A -85,B 0,C 180,E1 30947.223,E2 30947.223} C_VEL
LIN {X 0,Y 664.549,Z 178.383,A -85,B 0,C 180,E1 30944.327,E2 30944.327} C_VEL
LIN {X 0,Y 664.576,Z 178.377,A -85,B 0,C 180,E1 30941.667,E2 30941.667} C_VEL
LIN {X 0,Y 664.556,Z 178.378,A -85,B 0,C 180,E1 30938.554,E2 30938.554} C_VEL
LIN {X 0,Y 664.553,Z 178.383,A -85,B 0,C 180,E1 30936.031,E2 30936.031} C_VEL
LIN {X 0,Y 664.59,Z 178.364,A -85,B 0,C 180,E1 30932.976,E2 30932.976} C_VEL
LIN {X 0,Y 664.546,Z 178.373,A -85,B 0,C 180,E1 30930.329,E2 30930.329} C_VEL
LIN {X 0,Y 664.613,Z 178.384,A -85,B 0,C 180,E1 30927.553,E2 30927.553} C_VEL
LIN {X 0,Y 664.55,Z 178.375,A -85,B 0,C 180,E1 30924.6,E2 30924.6} C_VEL
LIN {X 0,Y 664.564,Z 178.384,A -85,B 0,C 180,E1 30922.021,E2 30922.021} C_VEL
LIN {X 0,Y 664.566,Z 178.383,A -85,B 0,C 180,E1 30918.89,E2 30918.89} C_VEL
LIN {X 0,Y 664.555,Z 178.38,A -85,B 0,C 180,E1 30916.229,E2 30916.229} C_VEL
LIN {X 0,Y 664.59,Z 178.379,A -85,B 0,C 180,E1 30913.193,E2 30913.193} C_VEL
LIN {X 0,Y 664.548,Z 178.387,A -85,B 0,C 180,E1 30910.534,E2 30910.534} C_VEL
LIN {X 0,Y 664.622,Z 178.345,A -85,B 0,C 180,E1 30907.689,E2 30907.689} C_VEL
LIN {X 0,Y 664.55,Z 178.385,A -85,B 0,C 180,E1 30904.762,E2 30904.762} C_VEL
LIN {X 0,Y 664.633,Z 178.566,A -85,B 0,C 180,E1 30903.417,E2 30903.417} C_VEL
LIN {X 0,Y 670.78,Z 199.313,A -85,B 0,C 180,E1 30901.243,E2 30901.243} C_VEL
LIN {X 0,Y 670.006,Z 225.856,A -85,B 0,C 180,E1 30899.027,E2 30899.027} C_VEL
LIN {X 0,Y 674.064,Z 244.564,A -85,B 0,C 180,E1 30898.612,E2 30898.612} C_VEL
LIN {X 0,Y 672.04,Z 515.437,A -85,B 0,C 180,E1 30895.523,E2 30895.523} C_VEL
LIN {X 0,Y 671.645,Z 539.176,A -85,B 0,C 180,E1 30895.177,E2 30895.177} C_VEL
LIN {X 0,Y 671.244,Z 557.369,A -85,B 0,C 180,E1 30894.791,E2 30894.791} C_VEL
LIN {X 0,Y 670.78,Z 574.145,A -85,B 0,C 180,E1 30894.337,E2 30894.337} C_VEL
LIN {X 0,Y 670.246,Z 590.507,A -85,B 0,C 180,E1 30893.796,E2 30893.796} C_VEL
LIN {X 0,Y 669.649,Z 606.545,A -85,B 0,C 180,E1 30893.166,E2 30893.166} C_VEL
LIN {X 0,Y 669.048,Z 622.226,A -85,B 0,C 180,E1 30892.445,E2 30892.445} C_VEL
LIN {X 0,Y 668.388,Z 638.303,A -85,B 0,C 180,E1 30891.59,E2 30891.59} C_VEL
LIN {X 0,Y 667.578,Z 657.229,A -85,B 0,C 180,E1 30890.422,E2 30890.422} C_VEL
LIN {X 0,Y 666.794,Z 674.672,A -85,B 0,C 180,E1 30889.14,E2 30889.14} C_VEL
LIN {X 0,Y 666.188,Z 688.656,A -85,B 0,C 180,E1 30887.963,E2 30887.963} C_VEL
LIN {X 0,Y 665.64,Z 702.148,A -85,B 0,C 180,E1 30886.671,E2 30886.671} C_VEL
LIN {X 0,Y 665.109,Z 716.636,A -85,B 0,C 180,E1 30885.073,E2 30885.073} C_VEL
LIN {X 0,Y 664.673,Z 729.431,A -85,B 0,C 180,E1 30883.393,E2 30883.393} C_VEL
LIN {X 0,Y 664.379,Z 739.762,A -85,B 0,C 180,E1 30881.809,E2 30881.809} C_VEL
LIN {X 0,Y 664.164,Z 749.867,A -85,B 0,C 180,E1 30879.969,E2 30879.969} C_VEL
LIN {X 0,Y 664.028,Z 757.869,A -85,B 0,C 180,E1 30878.136,E2 30878.136} C_VEL
LIN {X 0,Y 663.955,Z 763.876,A -85,B 0,C 180,E1 30876.398,E2 30876.398} C_VEL
LIN {X 0,Y 663.916,Z 768.398,A -85,B 0,C 180,E1 30874.664,E2 30874.664} C_VEL
LIN {X 0,Y 663.912,Z 771.917,A -85,B 0,C 180,E1 30872.589,E2 30872.589} C_VEL
LIN {X 0,Y 663.909,Z 773.278,A -85,B 0,C 180,E1 30870.777,E2 30870.777} C_VEL
LIN {X 0,Y 663.911,Z 773.249,A -85,B 0,C 180,E1 30869.137,E2 30869.137} C_VEL
LIN {X 0,Y 663.911,Z 771.825,A -85,B 0,C 180,E1 30867.324,E2 30867.324} C_VEL
LIN {X 0,Y 663.916,Z 768.398,A -85,B 0,C 180,E1 30865.336,E2 30865.336} C_VEL
LIN {X 0,Y 663.955,Z 763.876,A -85,B 0,C 180,E1 30863.602,E2 30863.602} C_VEL
LIN {X 0,Y 664.028,Z 757.869,A -85,B 0,C 180,E1 30861.864,E2 30861.864} C_VEL
LIN {X 0,Y 664.173,Z 749.426,A -85,B 0,C 180,E1 30859.944,E2 30859.944} C_VEL
LIN {X 0,Y 664.379,Z 739.762,A -85,B 0,C 180,E1 30858.191,E2 30858.191} C_VEL
LIN {X 0,Y 664.654,Z 730.045,A -85,B 0,C 180,E1 30856.695,E2 30856.695} C_VEL
LIN {X 0,Y 665.024,Z 718.728,A -85,B 0,C 180,E1 30855.191,E2 30855.191} C_VEL
LIN {X 0,Y 665.606,Z 703.033,A -85,B 0,C 180,E1 30853.418,E2 30853.418} C_VEL
LIN {X 0,Y 666.17,Z 689.153,A -85,B 0,C 180,E1 30852.082,E2 30852.082} C_VEL
LIN {X 0,Y 666.757,Z 675.43,A -85,B 0,C 180,E1 30850.921,E2 30850.921} C_VEL
LIN {X 0,Y 667.489,Z 659.145,A -85,B 0,C 180,E1 30849.712,E2 30849.712} C_VEL
LIN {X 0,Y 668.326,Z 639.909,A -85,B 0,C 180,E1 30848.5,E2 30848.5} C_VEL
LIN {X 0,Y 669.016,Z 623.143,A -85,B 0,C 180,E1 30847.6,E2 30847.6} C_VEL
LIN {X 0,Y 669.608,Z 607.604,A -85,B 0,C 180,E1 30846.879,E2 30846.879} C_VEL
LIN {X 0,Y 670.201,Z 591.748,A -85,B 0,C 180,E1 30846.249,E2 30846.249} C_VEL
LIN {X 0,Y 670.73,Z 575.631,A -85,B 0,C 180,E1 30845.708,E2 30845.708} C_VEL
LIN {X 0,Y 671.213,Z 558.627,A -85,B 0,C 180,E1 30845.24,E2 30845.24} C_VEL
LIN {X 0,Y 671.597,Z 541.682,A -85,B 0,C 180,E1 30844.871,E2 30844.871} C_VEL
LIN {X 0,Y 671.906,Z 523.964,A -85,B 0,C 180,E1 30844.587,E2 30844.587} C_VEL
LIN {X 0,Y 673.939,Z 261.262,A -85,B 0,C 180,E1 30841.581,E2 30841.581} C_VEL
LIN {X 0,Y 673.886,Z 242.916,A -85,B 0,C 180,E1 30841.361,E2 30841.361} C_VEL
LIN {X 0,Y 669.962,Z 225.312,A -85,B 0,C 180,E1 30840.945,E2 30840.945} C_VEL
LIN {X 0,Y 670.78,Z 199.313,A -85,B 0,C 180,E1 30838.757,E2 30838.757} C_VEL
LIN {X 0,Y 664.628,Z 178.521,A -85,B 0,C 180,E1 30836.57,E2 30836.57} C_VEL
LIN {X 0,Y 664.551,Z 178.369,A -85,B 0,C 180,E1 30833.607,E2 30833.607} C_VEL
LIN {X 0,Y 664.572,Z 178.37,A -85,B 0,C 180,E1 30830.926,E2 30830.926} C_VEL
LIN {X 0,Y 664.562,Z 178.379,A -85,B 0,C 180,E1 30827.859,E2 30827.859} C_VEL
LIN {X 0,Y 664.554,Z 178.383,A -85,B 0,C 180,E1 30825.247,E2 30825.247} C_VEL
LIN {X 0,Y 664.601,Z 178.383,A -85,B 0,C 180,E1 30822.259,E2 30822.259} C_VEL
LIN {X 0,Y 664.547,Z 178.375,A -85,B 0,C 180,E1 30819.528,E2 30819.528} C_VEL
LIN {X 0,Y 664.626,Z 178.38,A -85,B 0,C 180,E1 30816.674,E2 30816.674} C_VEL
LIN {X 0,Y 664.547,Z 178.379,A -85,B 0,C 180,E1 30813.701,E2 30813.701} C_VEL
LIN {X 0,Y 664.593,Z 178.383,A -85,B 0,C 180,E1 30810.967,E2 30810.967} C_VEL
LIN {X 0,Y 664.555,Z 178.364,A -85,B 0,C 180,E1 30807.984,E2 30807.984} C_VEL
LIN {X 0,Y 664.558,Z 178.38,A -85,B 0,C 180,E1 30805.392,E2 30805.392} C_VEL
LIN {X 0,Y 664.575,Z 178.377,A -85,B 0,C 180,E1 30802.281,E2 30802.281} C_VEL
LIN {X 0,Y 664.547,Z 178.383,A -85,B 0,C 180,E1 30799.65,E2 30799.65} C_VEL
LIN {X 0,Y 664.622,Z 178.378,A -85,B 0,C 180,E1 30796.699,E2 30796.699} C_VEL
LIN {X 0,Y 664.547,Z 178.379,A -85,B 0,C 180,E1 30793.93,E2 30793.93} C_VEL
LIN {X 0,Y 664.591,Z 178.379,A -85,B 0,C 180,E1 30791.191,E2 30791.191} C_VEL
LIN {X 0,Y 664.552,Z 178.375,A -85,B 0,C 180,E1 30788.152,E2 30788.152} C_VEL
LIN {X 0,Y 664.551,Z 178.383,A -85,B 0,C 180,E1 30785.699,E2 30785.699} C_VEL
LIN {X 0,Y 664.595,Z 178.38,A -85,B 0,C 180,E1 30782.673,E2 30782.673} C_VEL
LIN {X 0,Y 664.546,Z 178.383,A -85,B 0,C 180,E1 30780,E2 30780} C_VEL
LIN {X 0,Y 664.605,Z 178.375,A -85,B 0,C 180,E1 30777.241,E2 30777.241} C_VEL
LIN {X 0,Y 664.55,Z 178.381,A -85,B 0,C 180,E1 30774.301,E2 30774.301} C_VEL
LIN {X 0,Y 664.554,Z 178.379,A -85,B 0,C 180,E1 30771.782,E2 30771.782} C_VEL
LIN {X 0,Y 664.581,Z 178.377,A -85,B 0,C 180,E1 30768.721,E2 30768.721} C_VEL
LIN {X 0,Y 664.547,Z 178.383,A -85,B 0,C 180,E1 30766.012,E2 30766.012} C_VEL
LIN {X 0,Y 664.623,Z 178.376,A -85,B 0,C 180,E1 30763.077,E2 30763.077} C_VEL
LIN {X 0,Y 664.546,Z 178.383,A -85,B 0,C 180,E1 30760.212,E2 30760.212} C_VEL
LIN {X 0,Y 664.625,Z 178.378,A -85,B 0,C 180,E1 30757.348,E2 30757.348} C_VEL
LIN {X 0,Y 664.548,Z 178.377,A -85,B 0,C 180,E1 30754.416,E2 30754.416} C_VEL
LIN {X 0,Y 664.579,Z 178.357,A -85,B 0,C 180,E1 30751.71,E2 30751.71} C_VEL
LIN {X 0,Y 664.558,Z 178.384,A -85,B 0,C 180,E1 30748.704,E2 30748.704} C_VEL
LIN {X 0,Y 664.553,Z 178.377,A -85,B 0,C 180,E1 30746.068,E2 30746.068} C_VEL
LIN {X 0,Y 664.625,Z 178.37,A -85,B 0,C 180,E1 30743.39,E2 30743.39} C_VEL
LIN {X 0,Y 663.619,Z 178.506,A -85,B 0,C 180,E1 30742.726,E2 30742.726} C_VEL
LIN {X 0,Y 657.145,Z 179.31,A -85,B 0,C 180,E1 30740.865,E2 30740.865} C_VEL
LIN {X 0,Y 656.608,Z 179.373,A -85,B 0,C 180,E1 30740.38,E2 30740.38} C_VEL
LIN {X 0,Y 656.681,Z 179.373,A -85,B 0,C 180,E1 30737.582,E2 30737.582} C_VEL
LIN {X 0,Y 656.61,Z 179.374,A -85,B 0,C 180,E1 30734.671,E2 30734.671} C_VEL
LIN {X 0,Y 656.64,Z 179.373,A -85,B 0,C 180,E1 30731.943,E2 30731.943} C_VEL
LIN {X 0,Y 656.615,Z 179.374,A -85,B 0,C 180,E1 30728.852,E2 30728.852} C_VEL
LIN {X 0,Y 656.624,Z 179.373,A -85,B 0,C 180,E1 30726.189,E2 30726.189} C_VEL
LIN {X 0,Y 656.623,Z 179.374,A -85,B 0,C 180,E1 30723.03,E2 30723.03} C_VEL
LIN {X 0,Y 656.616,Z 179.373,A -85,B 0,C 180,E1 30720.364,E2 30720.364} C_VEL
LIN {X 0,Y 656.641,Z 179.373,A -85,B 0,C 180,E1 30717.276,E2 30717.276} C_VEL
LIN {X 0,Y 656.61,Z 179.375,A -85,B 0,C 180,E1 30714.561,E2 30714.561} C_VEL
LIN {X 0,Y 656.679,Z 179.372,A -85,B 0,C 180,E1 30711.619,E2 30711.619} C_VEL
LIN {X 0,Y 656.608,Z 179.375,A -85,B 0,C 180,E1 30708.832,E2 30708.832} C_VEL
LIN {X 0,Y 656.686,Z 179.372,A -85,B 0,C 180,E1 30705.905,E2 30705.905} C_VEL
LIN {X 0,Y 656.608,Z 179.374,A -85,B 0,C 180,E1 30702.94,E2 30702.94} C_VEL
LIN {X 0,Y 656.669,Z 179.372,A -85,B 0,C 180,E1 30700.083,E2 30700.083} C_VEL
LIN {X 0,Y 656.613,Z 179.376,A -85,B 0,C 180,E1 30697.172,E2 30697.172} C_VEL
LIN {X 0,Y 656.623,Z 179.375,A -85,B 0,C 180,E1 30694.541,E2 30694.541} C_VEL
LIN {X 0,Y 656.622,Z 179.375,A -85,B 0,C 180,E1 30691.396,E2 30691.396} C_VEL
